LIN {X 0,Y 421.12,Z 160.701,A -85,B 0,C 180,E1 -10145.341,E2 -10145.341} C_VEL
LIN {X 0,Y 421.143,Z 165.944,A -85,B 0,C 180,E1 -10146.39,E2 -10146.39} C_VEL
LIN {X 0,Y 419.835,Z 185.67,A -85,B 0,C 180,E1 -10150.217,E2 -10150.217} C_VEL
LIN {X 0,Y 419.588,Z 189.326,A -85,B 0,C 180,E1 -10150.921,E2 -10150.921} C_VEL
LIN {X 0,Y 423.684,Z 215.471,A -85,B 0,C 180,E1 -10151.572,E2 -10151.572} C_VEL
LIN {X 0,Y 422.852,Z 297.887,A -85,B 0,C 180,E1 -10152.997,E2 -10152.997} C_VEL
LIN {X 0,Y 422.296,Z 311.131,A -85,B 0,C 180,E1 -10153.41,E2 -10153.41} C_VEL
LIN {X 0,Y 421.611,Z 324.403,A -85,B 0,C 180,E1 -10154.035,E2 -10154.035} C_VEL
LIN {X 0,Y 420.908,Z 335.549,A -85,B 0,C 180,E1 -10154.753,E2 -10154.753} C_VEL
LIN {X 0,Y 420.13,Z 347.243,A -85,B 0,C 180,E1 -10155.724,E2 -10155.724} C_VEL
LIN {X 0,Y 419.409,Z 357.602,A -85,B 0,C 180,E1 -10156.802,E2 -10156.802} C_VEL
LIN {X 0,Y 418.836,Z 366.15,A -85,B 0,C 180,E1 -10157.892,E2 -10157.892} C_VEL
LIN {X 0,Y 418.209,Z 374.037,A -85,B 0,C 180,E1 -10159.102,E2 -10159.102} C_VEL
LIN {X 0,Y 417.71,Z 381.744,A -85,B 0,C 180,E1 -10160.558,E2 -10160.558} C_VEL
LIN {X 0,Y 417.328,Z 388.855,A -85,B 0,C 180,E1 -10162.257,E2 -10162.257} C_VEL
LIN {X 0,Y 417.119,Z 393.75,A -85,B 0,C 180,E1 -10163.767,E2 -10163.767} C_VEL
LIN {X 0,Y 417.102,Z 397.206,A -85,B 0,C 180,E1 -10165.167,E2 -10165.167} C_VEL
LIN {X 0,Y 417.015,Z 399.07,A -85,B 0,C 180,E1 -10166.134,E2 -10166.134} C_VEL
LIN {X 0,Y 417.032,Z 400.471,A -85,B 0,C 180,E1 -10167.102,E2 -10167.102} C_VEL
LIN {X 0,Y 417.07,Z 401.471,A -85,B 0,C 180,E1 -10168.068,E2 -10168.068} C_VEL
LIN {X 0,Y 417.034,Z 402.08,A -85,B 0,C 180,E1 -10169.034,E2 -10169.034} C_VEL
LIN {X 0,Y 417.031,Z 402.296,A -85,B 0,C 180,E1 -10169.999,E2 -10169.999} C_VEL
LIN {X 0,Y 417.069,Z 401.469,A -85,B 0,C 180,E1 -10171.931,E2 -10171.931} C_VEL
LIN {X 0,Y 417.031,Z 400.469,A -85,B 0,C 180,E1 -10172.897,E2 -10172.897} C_VEL
LIN {X 0,Y 417.015,Z 399.066,A -85,B 0,C 180,E1 -10173.865,E2 -10173.865} C_VEL
LIN {X 0,Y 417.115,Z 396.122,A -85,B 0,C 180,E1 -10175.317,E2 -10175.317} C_VEL
LIN {X 0,Y 417.231,Z 392.136,A -85,B 0,C 180,E1 -10176.771,E2 -10176.771} C_VEL
LIN {X 0,Y 417.485,Z 386.009,A -85,B 0,C 180,E1 -10178.47,E2 -10178.47} C_VEL
LIN {X 0,Y 417.873,Z 379.318,A -85,B 0,C 180,E1 -10179.926,E2 -10179.926} C_VEL
LIN {X 0,Y 418.438,Z 371.019,A -85,B 0,C 180,E1 -10181.381,E2 -10181.381} C_VEL
LIN {X 0,Y 419.083,Z 362.518,A -85,B 0,C 180,E1 -10182.591,E2 -10182.591} C_VEL
LIN {X 0,Y 419.803,Z 352.477,A -85,B 0,C 180,E1 -10183.752,E2 -10183.752} C_VEL
LIN {X 0,Y 420.497,Z 341.624,A -85,B 0,C 180,E1 -10184.766,E2 -10184.766} C_VEL
LIN {X 0,Y 421.248,Z 330.238,A -85,B 0,C 180,E1 -10185.606,E2 -10185.606} C_VEL
LIN {X 0,Y 421.911,Z 318.552,A -85,B 0,C 180,E1 -10186.263,E2 -10186.263} C_VEL
LIN {X 0,Y 422.541,Z 306.004,A -85,B 0,C 180,E1 -10186.766,E2 -10186.766} C_VEL
LIN {X 0,Y 422.933,Z 293.279,A -85,B 0,C 180,E1 -10187.092,E2 -10187.092} C_VEL
LIN {X 0,Y 423.594,Z 214.784,A -85,B 0,C 180,E1 -10188.436,E2 -10188.436} C_VEL
LIN {X 0,Y 419.587,Z 189.324,A -85,B 0,C 180,E1 -10189.072,E2 -10189.072} C_VEL
LIN {X 0,Y 420.757,Z 171.129,A -85,B 0,C 180,E1 -10192.592,E2 -10192.592} C_VEL
LIN {X 0,Y 421.281,Z 161.977,A -85,B 0,C 180,E1 -10194.386,E2 -10194.386} C_VEL
LIN {X 0,Y 419.312,Z 151.398,A -85,B 0,C 180,E1 -10196.637,E2 -10196.637} C_VEL
LIN {X 0,Y 418.285,Z 146.379,A -85,B 0,C 180,E1 -10197.751,E2 -10197.751} C_VEL
LIN {X 0,Y 418.236,Z 146.389,A -85,B 0,C 180,E1 -10201.018,E2 -10201.018} C_VEL
LIN {X 0,Y 418.229,Z 146.39,A -85,B 0,C 180,E1 -10203.678,E2 -10203.678} C_VEL
LIN {X 0,Y 418.234,Z 146.389,A -85,B 0,C 180,E1 -10207.223,E2 -10207.223} C_VEL
LIN {X 0,Y 418.203,Z 146.39,A -85,B 0,C 180,E1 -10210.866,E2 -10210.866} C_VEL
LIN {X 0,Y 418.199,Z 146.39,A -85,B 0,C 180,E1 -10213.728,E2 -10213.728} C_VEL
LIN {X 0,Y 418.194,Z 146.389,A -85,B 0,C 180,E1 -10216.447,E2 -10216.447} C_VEL
LIN {X 0,Y 418.204,Z 146.395,A -85,B 0,C 180,E1 -10219.131,E2 -10219.131} C_VEL
LIN {X 0,Y 418.231,Z 146.389,A -85,B 0,C 180,E1 -10222.775,E2 -10222.775} C_VEL
LIN {X 0,Y 418.225,Z 146.386,A -85,B 0,C 180,E1 -10226.321,E2 -10226.321} C_VEL
LIN {X 0,Y 418.231,Z 146.384,A -85,B 0,C 180,E1 -10229.727,E2 -10229.727} C_VEL
LIN {X 0,Y 418.203,Z 146.392,A -85,B 0,C 180,E1 -10233.016,E2 -10233.016} C_VEL
LIN {X 0,Y 418.249,Z 146.385,A -85,B 0,C 180,E1 -10236.216,E2 -10236.216} C_VEL
LIN {X 0,Y 418.237,Z 146.384,A -85,B 0,C 180,E1 -10239.336,E2 -10239.336} C_VEL
LIN {X 0,Y 418.237,Z 146.39,A -85,B 0,C 180,E1 -10242.394,E2 -10242.394} C_VEL
LIN {X 0,Y 418.267,Z 146.38,A -85,B 0,C 180,E1 -10245.402,E2 -10245.402} C_VEL
LIN {X 0,Y 418.292,Z 146.383,A -85,B 0,C 180,E1 -10248.368,E2 -10248.368} C_VEL
LIN {X 0,Y 418.436,Z 146.365,A -85,B 0,C 180,E1 -10252.278,E2 -10252.278} C_VEL
LIN {X 0,Y 418.458,Z 146.362,A -85,B 0,C 180,E1 -10254.217,E2 -10254.217} C_VEL
LIN {X 0,Y 418.522,Z 146.355,A -85,B 0,C 180,E1 -10258.075,E2 -10258.075} C_VEL
LIN {X 0,Y 418.396,Z 146.364,A -85,B 0,C 180,E1 -10260.963,E2 -10260.963} C_VEL
LIN {X 0,Y 418.459,Z 146.356,A -85,B 0,C 180,E1 -10262.888,E2 -10262.888} C_VEL
LIN {X 0,Y 418.432,Z 146.36,A -85,B 0,C 180,E1 -10266.46,E2 -10266.46} C_VEL
LIN {X 0,Y 418.367,Z 146.367,A -85,B 0,C 180,E1 -10268.696,E2 -10268.696} C_VEL
LIN {X 0,Y 418.304,Z 146.383,A -85,B 0,C 180,E1 -10271.631,E2 -10271.631} C_VEL
LIN {X 0,Y 418.268,Z 146.38,A -85,B 0,C 180,E1 -10274.598,E2 -10274.598} C_VEL
LIN {X 0,Y 418.246,Z 146.388,A -85,B 0,C 180,E1 -10277.606,E2 -10277.606} C_VEL
LIN {X 0,Y 418.24,Z 146.384,A -85,B 0,C 180,E1 -10280.664,E2 -10280.664} C_VEL
LIN {X 0,Y 418.25,Z 146.384,A -85,B 0,C 180,E1 -10283.784,E2 -10283.784} C_VEL
LIN {X 0,Y 418.21,Z 146.392,A -85,B 0,C 180,E1 -10287.046,E2 -10287.046} C_VEL
LIN {X 0,Y 418.234,Z 146.384,A -85,B 0,C 180,E1 -10290.273,E2 -10290.273} C_VEL
LIN {X 0,Y 418.226,Z 146.386,A -85,B 0,C 180,E1 -10293.679,E2 -10293.679} C_VEL
LIN {X 0,Y 418.233,Z 146.388,A -85,B 0,C 180,E1 -10297.225,E2 -10297.225} C_VEL
LIN {X 0,Y 418.205,Z 146.394,A -85,B 0,C 180,E1 -10300.869,E2 -10300.869} C_VEL
LIN {X 0,Y 418.199,Z 146.388,A -85,B 0,C 180,E1 -10303.729,E2 -10303.729} C_VEL
LIN {X 0,Y 418.203,Z 146.392,A -85,B 0,C 180,E1 -10306.449,E2 -10306.449} C_VEL
LIN {X 0,Y 418.213,Z 146.388,A -85,B 0,C 180,E1 -10309.132,E2 -10309.132} C_VEL
LIN {X 0,Y 418.218,Z 146.389,A -85,B 0,C 180,E1 -10312.169,E2 -10312.169} C_VEL
LIN {X 0,Y 418.263,Z 146.38,A -85,B 0,C 180,E1 -10315.421,E2 -10315.421} C_VEL
LIN {X 0,Y 418.21,Z 146.391,A -85,B 0,C 180,E1 -10318.605,E2 -10318.605} C_VEL
LIN {X 0,Y 418.241,Z 146.387,A -85,B 0,C 180,E1 -10321.934,E2 -10321.934} C_VEL
LIN {X 0,Y 418.253,Z 146.382,A -85,B 0,C 180,E1 -10325.161,E2 -10325.161} C_VEL
LIN {X 0,Y 418.274,Z 146.556,A -85,B 0,C 180,E1 -10327.66,E2 -10327.66} C_VEL
LIN {X 0,Y 420.194,Z 156.495,A -85,B 0,C 180,E1 -10330.03,E2 -10330.03} C_VEL
LIN {X 0,Y 420.055,Z 160.959,A -85,B 0,C 180,E1 -10331.01,E2 -10331.01} C_VEL
LIN {X 0,Y 424.093,Z 181.216,A -85,B 0,C 180,E1 -10331.558,E2 -10331.558} C_VEL
LIN {X 0,Y 423.051,Z 267.557,A -85,B 0,C 180,E1 -10333.037,E2 -10333.037} C_VEL
LIN {X 0,Y 422.732,Z 281.057,A -85,B 0,C 180,E1 -10333.459,E2 -10333.459} C_VEL
LIN {X 0,Y 422.184,Z 293.856,A -85,B 0,C 180,E1 -10334.058,E2 -10334.058} C_VEL
LIN {X 0,Y 421.531,Z 305.213,A -85,B 0,C 180,E1 -10334.777,E2 -10334.777} C_VEL
LIN {X 0,Y 420.921,Z 316.902,A -85,B 0,C 180,E1 -10335.747,E2 -10335.747} C_VEL
LIN {X 0,Y 420.246,Z 327.312,A -85,B 0,C 180,E1 -10336.83,E2 -10336.83} C_VEL
LIN {X 0,Y 419.539,Z 335.854,A -85,B 0,C 180,E1 -10337.914,E2 -10337.914} C_VEL
LIN {X 0,Y 418.928,Z 343.718,A -85,B 0,C 180,E1 -10339.122,E2 -10339.122} C_VEL
LIN {X 0,Y 418.35,Z 351.403,A -85,B 0,C 180,E1 -10340.574,E2 -10340.574} C_VEL
LIN {X 0,Y 418.307,Z 351.96,A -85,B 0,C 180,E1 -10340.695,E2 -10340.695} C_VEL
LIN {X 0,Y 417.433,Z 355.07,A -85,B 0,C 180,E1 -10341.378,E2 -10341.378} C_VEL
LIN {X 0,Y 414.293,Z 359.681,A -85,B 0,C 180,E1 -10342.51,E2 -10342.51} C_VEL
LIN {X 0,Y 411.176,Z 363.603,A -85,B 0,C 180,E1 -10343.699,E2 -10343.699} C_VEL
LIN {X 0,Y 410.349,Z 365.616,A -85,B 0,C 180,E1 -10344.464,E2 -10344.464} C_VEL
LIN {X 0,Y 410.161,Z 368.857,A -85,B 0,C 180,E1 -10346.071,E2 -10346.071} C_VEL
LIN {X 0,Y 410.148,Z 370.254,A -85,B 0,C 180,E1 -10347.054,E2 -10347.054} C_VEL
LIN {X 0,Y 409.964,Z 371.864,A -85,B 0,C 180,E1 -10349.018,E2 -10349.018} C_VEL
LIN {X 0,Y 409.954,Z 372.098,A -85,B 0,C 180,E1 -10350.001,E2 -10350.001} C_VEL
LIN {X 0,Y 409.964,Z 371.91,A -85,B 0,C 180,E1 -10350.983,E2 -10350.983} C_VEL
LIN {X 0,Y 410.145,Z 370.359,A -85,B 0,C 180,E1 -10352.947,E2 -10352.947} C_VEL
LIN {X 0,Y 410.147,Z 369.009,A -85,B 0,C 180,E1 -10353.931,E2 -10353.931} C_VEL
LIN {X 0,Y 410.318,Z 366.15,A -85,B 0,C 180,E1 -10355.406,E2 -10355.406} C_VEL
LIN {X 0,Y 410.543,Z 362.273,A -85,B 0,C 180,E1 -10356.883,E2 -10356.883} C_VEL
LIN {X 0,Y 410.868,Z 357.269,A -85,B 0,C 180,E1 -10358.361,E2 -10358.361} C_VEL
LIN {X 0,Y 411.439,Z 350.965,A -85,B 0,C 180,E1 -10359.836,E2 -10359.836} C_VEL
LIN {X 0,Y 412.059,Z 343.075,A -85,B 0,C 180,E1 -10361.312,E2 -10361.312} C_VEL
LIN {X 0,Y 412.689,Z 335.03,A -85,B 0,C 180,E1 -10362.541,E2 -10362.541} C_VEL
LIN {X 0,Y 413.578,Z 325.204,A -85,B 0,C 180,E1 -10363.763,E2 -10363.763} C_VEL
LIN {X 0,Y 414.261,Z 314.161,A -85,B 0,C 180,E1 -10364.869,E2 -10364.869} C_VEL
LIN {X 0,Y 414.933,Z 303.326,A -85,B 0,C 180,E1 -10365.724,E2 -10365.724} C_VEL
LIN {X 0,Y 415.547,Z 291.357,A -85,B 0,C 180,E1 -10366.457,E2 -10366.457} C_VEL
LIN {X 0,Y 416.066,Z 278.207,A -85,B 0,C 180,E1 -10367.036,E2 -10367.036} C_VEL
LIN {X 0,Y 416.484,Z 264.956,A -85,B 0,C 180,E1 -10367.398,E2 -10367.398} C_VEL
LIN {X 0,Y 417.353,Z 181.348,A -85,B 0,C 180,E1 -10368.852,E2 -10368.852} C_VEL
LIN {X 0,Y 413.161,Z 161.121,A -85,B 0,C 180,E1 -10369.44,E2 -10369.44} C_VEL
LIN {X 0,Y 413.177,Z 157.551,A -85,B 0,C 180,E1 -10370.242,E2 -10370.242} C_VEL
LIN {X 0,Y 411.205,Z 147.261,A -85,B 0,C 180,E1 -10372.755,E2 -10372.755} C_VEL
LIN {X 0,Y 411.199,Z 147.263,A -85,B 0,C 180,E1 -10375.296,E2 -10375.296} C_VEL
LIN {X 0,Y 411.196,Z 147.261,A -85,B 0,C 180,E1 -10378.592,E2 -10378.592} C_VEL
LIN {X 0,Y 411.168,Z 147.268,A -85,B 0,C 180,E1 -10381.997,E2 -10381.997} C_VEL
LIN {X 0,Y 411.212,Z 147.259,A -85,B 0,C 180,E1 -10384.878,E2 -10384.878} C_VEL
LIN {X 0,Y 411.196,Z 147.262,A -85,B 0,C 180,E1 -10388.166,E2 -10388.166} C_VEL
LIN {X 0,Y 411.17,Z 147.267,A -85,B 0,C 180,E1 -10391.806,E2 -10391.806} C_VEL
LIN {X 0,Y 411.176,Z 147.268,A -85,B 0,C 180,E1 -10395.509,E2 -10395.509} C_VEL
LIN {X 0,Y 411.154,Z 147.268,A -85,B 0,C 180,E1 -10398.773,E2 -10398.773} C_VEL
LIN {X 0,Y 411.186,Z 147.262,A -85,B 0,C 180,E1 -10402.025,E2 -10402.025} C_VEL
LIN {X 0,Y 411.191,Z 147.262,A -85,B 0,C 180,E1 -10405.665,E2 -10405.665} C_VEL
LIN {X 0,Y 411.186,Z 147.267,A -85,B 0,C 180,E1 -10409.152,E2 -10409.152} C_VEL
LIN {X 0,Y 411.178,Z 147.265,A -85,B 0,C 180,E1 -10411.407,E2 -10411.407} C_VEL
LIN {X 0,Y 411.225,Z 147.263,A -85,B 0,C 180,E1 -10414.929,E2 -10414.929} C_VEL
LIN {X 0,Y 411.203,Z 147.26,A -85,B 0,C 180,E1 -10417.913,E2 -10417.913} C_VEL
LIN {X 0,Y 411.212,Z 147.261,A -85,B 0,C 180,E1 -10421.051,E2 -10421.051} C_VEL
LIN {X 0,Y 411.208,Z 147.262,A -85,B 0,C 180,E1 -10424.13,E2 -10424.13} C_VEL
LIN {X 0,Y 411.301,Z 147.248,A -85,B 0,C 180,E1 -10427.165,E2 -10427.165} C_VEL
LIN {X 0,Y 411.285,Z 147.254,A -85,B 0,C 180,E1 -10430.161,E2 -10430.161} C_VEL
LIN {X 0,Y 411.387,Z 147.237,A -85,B 0,C 180,E1 -10433.132,E2 -10433.132} C_VEL
LIN {X 0,Y 411.281,Z 147.25,A -85,B 0,C 180,E1 -10435.099,E2 -10435.099} C_VEL
LIN {X 0,Y 411.498,Z 147.229,A -85,B 0,C 180,E1 -10438.042,E2 -10438.042} C_VEL
LIN {X 0,Y 411.373,Z 147.239,A -85,B 0,C 180,E1 -10440.979,E2 -10440.979} C_VEL
LIN {X 0,Y 411.422,Z 147.233,A -85,B 0,C 180,E1 -10442.937,E2 -10442.937} C_VEL
LIN {X 0,Y 411.386,Z 147.237,A -85,B 0,C 180,E1 -10446.868,E2 -10446.868} C_VEL
LIN {X 0,Y 411.27,Z 147.258,A -85,B 0,C 180,E1 -10449.839,E2 -10449.839} C_VEL
LIN {X 0,Y 411.297,Z 147.249,A -85,B 0,C 180,E1 -10453.1,E2 -10453.1} C_VEL
LIN {X 0,Y 411.204,Z 147.26,A -85,B 0,C 180,E1 -10456.891,E2 -10456.891} C_VEL
LIN {X 0,Y 411.201,Z 147.262,A -85,B 0,C 180,E1 -10459.988,E2 -10459.988} C_VEL
LIN {X 0,Y 411.182,Z 147.266,A -85,B 0,C 180,E1 -10463.149,E2 -10463.149} C_VEL
LIN {X 0,Y 411.168,Z 147.264,A -85,B 0,C 180,E1 -10466.386,E2 -10466.386} C_VEL
LIN {X 0,Y 411.19,Z 147.263,A -85,B 0,C 180,E1 -10469.714,E2 -10469.714} C_VEL
LIN {X 0,Y 411.202,Z 147.267,A -85,B 0,C 180,E1 -10473.156,E2 -10473.156} C_VEL
LIN {X 0,Y 411.19,Z 147.263,A -85,B 0,C 180,E1 -10476.552,E2 -10476.552} C_VEL
LIN {X 0,Y 411.177,Z 147.263,A -85,B 0,C 180,E1 -10479.722,E2 -10479.722} C_VEL
LIN {X 0,Y 411.161,Z 147.269,A -85,B 0,C 180,E1 -10483.135,E2 -10483.135} C_VEL
LIN {X 0,Y 411.163,Z 147.265,A -85,B 0,C 180,E1 -10485.882,E2 -10485.882} C_VEL
LIN {X 0,Y 411.158,Z 147.266,A -85,B 0,C 180,E1 -10489.493,E2 -10489.493} C_VEL
LIN {X 0,Y 411.186,Z 147.263,A -85,B 0,C 180,E1 -10492.025,E2 -10492.025} C_VEL
LIN {X 0,Y 411.203,Z 147.261,A -85,B 0,C 180,E1 -10495.123,E2 -10495.123} C_VEL
LIN {X 0,Y 411.165,Z 147.267,A -85,B 0,C 180,E1 -10498.003,E2 -10498.003} C_VEL
LIN {X 0,Y 411.208,Z 147.263,A -85,B 0,C 180,E1 -10501.409,E2 -10501.409} C_VEL
LIN {X 0,Y 411.247,Z 147.354,A -85,B 0,C 180,E1 -10502.003,E2 -10502.003} C_VEL
LIN {X 0,Y 413.892,Z 160.426,A -85,B 0,C 180,E1 -10504.88,E2 -10504.88} C_VEL
LIN {X 0,Y 414.376,Z 164.377,A -85,B 0,C 180,E1 -10505.714,E2 -10505.714} C_VEL
LIN {X 0,Y 413.094,Z 182.725,A -85,B 0,C 180,E1 -10509.345,E2 -10509.345} C_VEL
LIN {X 0,Y 412.722,Z 188.983,A -85,B 0,C 180,E1 -10510.574,E2 -10510.574} C_VEL
LIN {X 0,Y 416.867,Z 215.868,A -85,B 0,C 180,E1 -10511.271,E2 -10511.271} C_VEL
LIN {X 0,Y 416.082,Z 297.641,A -85,B 0,C 180,E1 -10512.712,E2 -10512.712} C_VEL
LIN {X 0,Y 415.506,Z 310.88,A -85,B 0,C 180,E1 -10513.131,E2 -10513.131} C_VEL
LIN {X 0,Y 414.782,Z 324.149,A -85,B 0,C 180,E1 -10513.765,E2 -10513.765} C_VEL
LIN {X 0,Y 414.045,Z 335.293,A -85,B 0,C 180,E1 -10514.494,E2 -10514.494} C_VEL
LIN {X 0,Y 413.22,Z 346.897,A -85,B 0,C 180,E1 -10515.471,E2 -10515.471} C_VEL
LIN {X 0,Y 412.483,Z 357.345,A -85,B 0,C 180,E1 -10516.576,E2 -10516.576} C_VEL
LIN {X 0,Y 411.875,Z 365.893,A -85,B 0,C 180,E1 -10517.684,E2 -10517.684} C_VEL
LIN {X 0,Y 411.209,Z 373.778,A -85,B 0,C 180,E1 -10518.914,E2 -10518.914} C_VEL
LIN {X 0,Y 410.665,Z 381.485,A -85,B 0,C 180,E1 -10520.394,E2 -10520.394} C_VEL
LIN {X 0,Y 410.268,Z 388.596,A -85,B 0,C 180,E1 -10522.123,E2 -10522.123} C_VEL
LIN {X 0,Y 410.043,Z 393.819,A -85,B 0,C 180,E1 -10523.775,E2 -10523.775} C_VEL
LIN {X 0,Y 410.009,Z 396.947,A -85,B 0,C 180,E1 -10525.083,E2 -10525.083} C_VEL
LIN {X 0,Y 409.932,Z 398.812,A -85,B 0,C 180,E1 -10526.067,E2 -10526.067} C_VEL
LIN {X 0,Y 409.997,Z 401.213,A -85,B 0,C 180,E1 -10528.035,E2 -10528.035} C_VEL
LIN {X 0,Y 409.958,Z 401.821,A -85,B 0,C 180,E1 -10529.017,E2 -10529.017} C_VEL
LIN {X 0,Y 409.952,Z 402.037,A -85,B 0,C 180,E1 -10529.999,E2 -10529.999} C_VEL
LIN {X 0,Y 409.997,Z 401.211,A -85,B 0,C 180,E1 -10531.964,E2 -10531.964} C_VEL
LIN {X 0,Y 409.932,Z 398.806,A -85,B 0,C 180,E1 -10533.932,E2 -10533.932} C_VEL
LIN {X 0,Y 410.01,Z 395.861,A -85,B 0,C 180,E1 -10535.409,E2 -10535.409} C_VEL
LIN {X 0,Y 410.164,Z 391.876,A -85,B 0,C 180,E1 -10536.888,E2 -10536.888} C_VEL
LIN {X 0,Y 410.447,Z 385.748,A -85,B 0,C 180,E1 -10538.616,E2 -10538.616} C_VEL
LIN {X 0,Y 410.864,Z 379.056,A -85,B 0,C 180,E1 -10540.097,E2 -10540.097} C_VEL
LIN {X 0,Y 411.46,Z 370.757,A -85,B 0,C 180,E1 -10541.577,E2 -10541.577} C_VEL
LIN {X 0,Y 412.109,Z 362.254,A -85,B 0,C 180,E1 -10542.808,E2 -10542.808} C_VEL
LIN {X 0,Y 412.882,Z 351.988,A -85,B 0,C 180,E1 -10544.012,E2 -10544.012} C_VEL
LIN {X 0,Y 413.614,Z 341.36,A -85,B 0,C 180,E1 -10545.017,E2 -10545.017} C_VEL
LIN {X 0,Y 414.402,Z 329.974,A -85,B 0,C 180,E1 -10545.87,E2 -10545.87} C_VEL
LIN {X 0,Y 415.099,Z 318.286,A -85,B 0,C 180,E1 -10546.537,E2 -10546.537} C_VEL
LIN {X 0,Y 415.762,Z 305.736,A -85,B 0,C 180,E1 -10547.047,E2 -10547.047} C_VEL
LIN {X 0,Y 416.152,Z 293.003,A -85,B 0,C 180,E1 -10547.379,E2 -10547.379} C_VEL
LIN {X 0,Y 416.854,Z 215.725,A -85,B 0,C 180,E1 -10548.724,E2 -10548.724} C_VEL
LIN {X 0,Y 412.718,Z 189.239,A -85,B 0,C 180,E1 -10549.392,E2 -10549.392} C_VEL
LIN {X 0,Y 413.902,Z 170.865,A -85,B 0,C 180,E1 -10552.987,E2 -10552.987} C_VEL
LIN {X 0,Y 414.309,Z 163.019,A -85,B 0,C 180,E1 -10554.556,E2 -10554.556} C_VEL
LIN {X 0,Y 411.935,Z 150.593,A -85,B 0,C 180,E1 -10557.261,E2 -10557.261} C_VEL
LIN {X 0,Y 411.256,Z 147.256,A -85,B 0,C 180,E1 -10558.03,E2 -10558.03} C_VEL
LIN {X 0,Y 411.179,Z 147.269,A -85,B 0,C 180,E1 -10561.282,E2 -10561.282} C_VEL
LIN {X 0,Y 411.189,Z 147.262,A -85,B 0,C 180,E1 -10564.334,E2 -10564.334} C_VEL
LIN {X 0,Y 411.185,Z 147.263,A -85,B 0,C 180,E1 -10566.741,E2 -10566.741} C_VEL
LIN {X 0,Y 411.165,Z 147.268,A -85,B 0,C 180,E1 -10569.719,E2 -10569.719} C_VEL
LIN {X 0,Y 411.16,Z 147.271,A -85,B 0,C 180,E1 -10573.134,E2 -10573.134} C_VEL
LIN {X 0,Y 411.158,Z 147.266,A -85,B 0,C 180,E1 -10575.881,E2 -10575.881} C_VEL
LIN {X 0,Y 411.156,Z 147.268,A -85,B 0,C 180,E1 -10579.493,E2 -10579.493} C_VEL
LIN {X 0,Y 411.18,Z 147.263,A -85,B 0,C 180,E1 -10582.025,E2 -10582.025} C_VEL
LIN {X 0,Y 411.195,Z 147.266,A -85,B 0,C 180,E1 -10585.123,E2 -10585.123} C_VEL
LIN {X 0,Y 411.155,Z 147.266,A -85,B 0,C 180,E1 -10588.002,E2 -10588.002} C_VEL
LIN {X 0,Y 411.167,Z 147.265,A -85,B 0,C 180,E1 -10591.406,E2 -10591.406} C_VEL
LIN {X 0,Y 411.179,Z 147.267,A -85,B 0,C 180,E1 -10594.941,E2 -10594.941} C_VEL
LIN {X 0,Y 411.193,Z 147.262,A -85,B 0,C 180,E1 -10597.913,E2 -10597.913} C_VEL
LIN {X 0,Y 411.201,Z 147.262,A -85,B 0,C 180,E1 -10601.05,E2 -10601.05} C_VEL
LIN {X 0,Y 411.199,Z 147.264,A -85,B 0,C 180,E1 -10604.13,E2 -10604.13} C_VEL
LIN {X 0,Y 411.292,Z 147.249,A -85,B 0,C 180,E1 -10607.165,E2 -10607.165} C_VEL
LIN {X 0,Y 411.265,Z 147.258,A -85,B 0,C 180,E1 -10610.161,E2 -10610.161} C_VEL
LIN {X 0,Y 411.379,Z 147.238,A -85,B 0,C 180,E1 -10613.132,E2 -10613.132} C_VEL
LIN {X 0,Y 411.274,Z 147.251,A -85,B 0,C 180,E1 -10615.099,E2 -10615.099} C_VEL
LIN {X 0,Y 411.491,Z 147.231,A -85,B 0,C 180,E1 -10618.043,E2 -10618.043} C_VEL
LIN {X 0,Y 411.366,Z 147.24,A -85,B 0,C 180,E1 -10620.979,E2 -10620.979} C_VEL
LIN {X 0,Y 411.417,Z 147.233,A -85,B 0,C 180,E1 -10622.938,E2 -10622.938} C_VEL
LIN {X 0,Y 411.382,Z 147.238,A -85,B 0,C 180,E1 -10626.456,E2 -10626.456} C_VEL
LIN {X 0,Y 411.308,Z 147.247,A -85,B 0,C 180,E1 -10628.846,E2 -10628.846} C_VEL
LIN {X 0,Y 411.273,Z 147.256,A -85,B 0,C 180,E1 -10631.833,E2 -10631.833} C_VEL
LIN {X 0,Y 411.221,Z 147.258,A -85,B 0,C 180,E1 -10634.854,E2 -10634.854} C_VEL
LIN {X 0,Y 411.204,Z 147.262,A -85,B 0,C 180,E1 -10637.917,E2 -10637.917} C_VEL
LIN {X 0,Y 411.187,Z 147.265,A -85,B 0,C 180,E1 -10641.035,E2 -10641.035} C_VEL
LIN {X 0,Y 411.183,Z 147.262,A -85,B 0,C 180,E1 -10644.218,E2 -10644.218} C_VEL
LIN {X 0,Y 411.169,Z 147.268,A -85,B 0,C 180,E1 -10647.484,E2 -10647.484} C_VEL
LIN {X 0,Y 411.189,Z 147.263,A -85,B 0,C 180,E1 -10649.714,E2 -10649.714} C_VEL
LIN {X 0,Y 411.197,Z 147.266,A -85,B 0,C 180,E1 -10653.157,E2 -10653.157} C_VEL
LIN {X 0,Y 411.186,Z 147.265,A -85,B 0,C 180,E1 -10656.553,E2 -10656.553} C_VEL
LIN {X 0,Y 411.172,Z 147.264,A -85,B 0,C 180,E1 -10659.723,E2 -10659.723} C_VEL
LIN {X 0,Y 411.159,Z 147.268,A -85,B 0,C 180,E1 -10663.136,E2 -10663.136} C_VEL
LIN {X 0,Y 411.163,Z 147.265,A -85,B 0,C 180,E1 -10665.882,E2 -10665.882} C_VEL
LIN {X 0,Y 411.154,Z 147.271,A -85,B 0,C 180,E1 -10668.774,E2 -10668.774} C_VEL
LIN {X 0,Y 411.183,Z 147.264,A -85,B 0,C 180,E1 -10672.026,E2 -10672.026} C_VEL
LIN {X 0,Y 411.203,Z 147.26,A -85,B 0,C 180,E1 -10675.667,E2 -10675.667} C_VEL
LIN {X 0,Y 411.187,Z 147.262,A -85,B 0,C 180,E1 -10679.153,E2 -10679.153} C_VEL
LIN {X 0,Y 411.185,Z 147.266,A -85,B 0,C 180,E1 -10682.518,E2 -10682.518} C_VEL
LIN {X 0,Y 411.203,Z 147.263,A -85,B 0,C 180,E1 -10685.784,E2 -10685.784} C_VEL
LIN {X 0,Y 411.219,Z 147.419,A -85,B 0,C 180,E1 -10687.405,E2 -10687.405} C_VEL
LIN {X 0,Y 413.177,Z 157.134,A -85,B 0,C 180,E1 -10689.764,E2 -10689.764} C_VEL
LIN {X 0,Y 413.163,Z 161.186,A -85,B 0,C 180,E1 -10690.675,E2 -10690.675} C_VEL
LIN {X 0,Y 417.367,Z 181.958,A -85,B 0,C 180,E1 -10691.258,E2 -10691.258} C_VEL
LIN {X 0,Y 416.27,Z 267.835,A -85,B 0,C 180,E1 -10692.753,E2 -10692.753} C_VEL
LIN {X 0,Y 415.954,Z 281.326,A -85,B 0,C 180,E1 -10693.182,E2 -10693.182} C_VEL
LIN {X 0,Y 415.365,Z 294.123,A -85,B 0,C 180,E1 -10693.789,E2 -10693.789} C_VEL
LIN {X 0,Y 414.702,Z 305.478,A -85,B 0,C 180,E1 -10694.52,E2 -10694.52} C_VEL
LIN {X 0,Y 414.102,Z 316.122,A -85,B 0,C 180,E1 -10695.406,E2 -10695.406} C_VEL
LIN {X 0,Y 413.426,Z 326.511,A -85,B 0,C 180,E1 -10696.483,E2 -10696.483} C_VEL
LIN {X 0,Y 412.604,Z 336.116,A -85,B 0,C 180,E1 -10697.707,E2 -10697.707} C_VEL
LIN {X 0,Y 411.963,Z 343.98,A -85,B 0,C 180,E1 -10698.936,E2 -10698.936} C_VEL
LIN {X 0,Y 411.36,Z 351.664,A -85,B 0,C 180,E1 -10700.412,E2 -10700.412} C_VEL
LIN {X 0,Y 410.778,Z 358.714,A -85,B 0,C 180,E1 -10702.134,E2 -10702.134} C_VEL
LIN {X 0,Y 410.551,Z 363.004,A -85,B 0,C 180,E1 -10703.472,E2 -10703.472} C_VEL
LIN {X 0,Y 410.349,Z 365.616,A -85,B 0,C 180,E1 -10704.464,E2 -10704.464} C_VEL
LIN {X 0,Y 409.542,Z 367.409,A -85,B 0,C 180,E1 -10705.243,E2 -10705.243} C_VEL
LIN {X 0,Y 406.546,Z 369.725,A -85,B 0,C 180,E1 -10706.531,E2 -10706.531} C_VEL
LIN {X 0,Y 404.071,Z 371.118,A -85,B 0,C 180,E1 -10707.587,E2 -10707.587} C_VEL
LIN {X 0,Y 402.93,Z 371.908,A -85,B 0,C 180,E1 -10708.552,E2 -10708.552} C_VEL
LIN {X 0,Y 402.902,Z 371.933,A -85,B 0,C 180,E1 -10708.692,E2 -10708.692} C_VEL
LIN {X 0,Y 402.877,Z 372.356,A -85,B 0,C 180,E1 -10710.001,E2 -10710.001} C_VEL
LIN {X 0,Y 402.89,Z 372.168,A -85,B 0,C 180,E1 -10711,E2 -10711} C_VEL
LIN {X 0,Y 403.065,Z 370.618,A -85,B 0,C 180,E1 -10712.999,E2 -10712.999} C_VEL
LIN {X 0,Y 403.059,Z 369.268,A -85,B 0,C 180,E1 -10714,E2 -10714} C_VEL
LIN {X 0,Y 403.269,Z 366.407,A -85,B 0,C 180,E1 -10715.501,E2 -10715.501} C_VEL
LIN {X 0,Y 403.486,Z 362.531,A -85,B 0,C 180,E1 -10717.004,E2 -10717.004} C_VEL
LIN {X 0,Y 403.854,Z 357.527,A -85,B 0,C 180,E1 -10718.507,E2 -10718.507} C_VEL
LIN {X 0,Y 404.455,Z 351.222,A -85,B 0,C 180,E1 -10720.007,E2 -10720.007} C_VEL
LIN {X 0,Y 405.097,Z 343.332,A -85,B 0,C 180,E1 -10721.509,E2 -10721.509} C_VEL
LIN {X 0,Y 405.768,Z 335.286,A -85,B 0,C 180,E1 -10722.758,E2 -10722.758} C_VEL
LIN {X 0,Y 406.704,Z 325.459,A -85,B 0,C 180,E1 -10724.001,E2 -10724.001} C_VEL
LIN {X 0,Y 407.3,Z 315.798,A -85,B 0,C 180,E1 -10725.001,E2 -10725.001} C_VEL
LIN {X 0,Y 408.028,Z 305.336,A -85,B 0,C 180,E1 -10725.869,E2 -10725.869} C_VEL
LIN {X 0,Y 408.67,Z 293.859,A -85,B 0,C 180,E1 -10726.613,E2 -10726.613} C_VEL
LIN {X 0,Y 409.225,Z 280.878,A -85,B 0,C 180,E1 -10727.233,E2 -10727.233} C_VEL
LIN {X 0,Y 409.642,Z 268.165,A -85,B 0,C 180,E1 -10727.633,E2 -10727.633} C_VEL
LIN {X 0,Y 410.612,Z 182.102,A -85,B 0,C 180,E1 -10729.164,E2 -10729.164} C_VEL
LIN {X 0,Y 406.301,Z 161.329,A -85,B 0,C 180,E1 -10729.791,E2 -10729.791} C_VEL
LIN {X 0,Y 405.821,Z 156.281,A -85,B 0,C 180,E1 -10730.979,E2 -10730.979} C_VEL
LIN {X 0,Y 404.18,Z 148.135,A -85,B 0,C 180,E1 -10733.041,E2 -10733.041} C_VEL
LIN {X 0,Y 404.152,Z 148.144,A -85,B 0,C 180,E1 -10735.769,E2 -10735.769} C_VEL
LIN {X 0,Y 404.159,Z 148.138,A -85,B 0,C 180,E1 -10739.137,E2 -10739.137} C_VEL
LIN {X 0,Y 404.143,Z 148.139,A -85,B 0,C 180,E1 -10742.622,E2 -10742.622} C_VEL
LIN {X 0,Y 404.182,Z 148.137,A -85,B 0,C 180,E1 -10745.19,E2 -10745.19} C_VEL
LIN {X 0,Y 404.135,Z 148.141,A -85,B 0,C 180,E1 -10748.759,E2 -10748.759} C_VEL
LIN {X 0,Y 404.114,Z 148.148,A -85,B 0,C 180,E1 -10751.598,E2 -10751.598} C_VEL
LIN {X 0,Y 404.145,Z 148.139,A -85,B 0,C 180,E1 -10754.522,E2 -10754.522} C_VEL
LIN {X 0,Y 404.131,Z 148.148,A -85,B 0,C 180,E1 -10757.295,E2 -10757.295} C_VEL
LIN {X 0,Y 404.132,Z 148.141,A -85,B 0,C 180,E1 -10759.951,E2 -10759.951} C_VEL
LIN {X 0,Y 404.134,Z 148.148,A -85,B 0,C 180,E1 -10763.125,E2 -10763.125} C_VEL
LIN {X 0,Y 404.137,Z 148.14,A -85,B 0,C 180,E1 -10766.187,E2 -10766.187} C_VEL
LIN {X 0,Y 404.142,Z 148.14,A -85,B 0,C 180,E1 -10769.714,E2 -10769.714} C_VEL
LIN {X 0,Y 404.126,Z 148.145,A -85,B 0,C 180,E1 -10773.118,E2 -10773.118} C_VEL
LIN {X 0,Y 404.161,Z 148.14,A -85,B 0,C 180,E1 -10776.425,E2 -10776.425} C_VEL
LIN {X 0,Y 404.19,Z 148.134,A -85,B 0,C 180,E1 -10779.874,E2 -10779.874} C_VEL
LIN {X 0,Y 404.172,Z 148.138,A -85,B 0,C 180,E1 -10783.013,E2 -10783.013} C_VEL
LIN {X 0,Y 404.281,Z 148.124,A -85,B 0,C 180,E1 -10786.939,E2 -10786.939} C_VEL
LIN {X 0,Y 404.251,Z 148.129,A -85,B 0,C 180,E1 -10789.988,E2 -10789.988} C_VEL
LIN {X 0,Y 404.337,Z 148.116,A -85,B 0,C 180,E1 -10793.011,E2 -10793.011} C_VEL
LIN {X 0,Y 404.253,Z 148.126,A -85,B 0,C 180,E1 -10795.013,E2 -10795.013} C_VEL
LIN {X 0,Y 404.467,Z 148.104,A -85,B 0,C 180,E1 -10798.008,E2 -10798.008} C_VEL
LIN {X 0,Y 404.343,Z 148.114,A -85,B 0,C 180,E1 -10800.996,E2 -10800.996} C_VEL
LIN {X 0,Y 404.355,Z 148.113,A -85,B 0,C 180,E1 -10802.989,E2 -10802.989} C_VEL
LIN {X 0,Y 404.362,Z 148.118,A -85,B 0,C 180,E1 -10805.986,E2 -10805.986} C_VEL
LIN {X 0,Y 404.251,Z 148.126,A -85,B 0,C 180,E1 -10809.002,E2 -10809.002} C_VEL
LIN {X 0,Y 404.24,Z 148.131,A -85,B 0,C 180,E1 -10812.042,E2 -10812.042} C_VEL
LIN {X 0,Y 404.153,Z 148.14,A -85,B 0,C 180,E1 -10815.12,E2 -10815.12} C_VEL
LIN {X 0,Y 404.132,Z 148.141,A -85,B 0,C 180,E1 -10818.242,E2 -10818.242} C_VEL
LIN {X 0,Y 404.127,Z 148.148,A -85,B 0,C 180,E1 -10821.42,E2 -10821.42} C_VEL
LIN {X 0,Y 404.132,Z 148.141,A -85,B 0,C 180,E1 -10824.669,E2 -10824.669} C_VEL
LIN {X 0,Y 404.098,Z 148.145,A -85,B 0,C 180,E1 -10828.007,E2 -10828.007} C_VEL
LIN {X 0,Y 404.137,Z 148.14,A -85,B 0,C 180,E1 -10830.286,E2 -10830.286} C_VEL
LIN {X 0,Y 404.136,Z 148.141,A -85,B 0,C 180,E1 -10833.813,E2 -10833.813} C_VEL
LIN {X 0,Y 404.133,Z 148.146,A -85,B 0,C 180,E1 -10836.875,E2 -10836.875} C_VEL
LIN {X 0,Y 404.116,Z 148.143,A -85,B 0,C 180,E1 -10840.075,E2 -10840.075} C_VEL
LIN {X 0,Y 404.141,Z 148.144,A -85,B 0,C 180,E1 -10843.082,E2 -10843.082} C_VEL
LIN {X 0,Y 404.12,Z 148.142,A -85,B 0,C 180,E1 -10845.922,E2 -10845.922} C_VEL
LIN {X 0,Y 404.102,Z 148.151,A -85,B 0,C 180,E1 -10848.633,E2 -10848.633} C_VEL
LIN {X 0,Y 404.14,Z 148.14,A -85,B 0,C 180,E1 -10851.495,E2 -10851.495} C_VEL
LIN {X 0,Y 404.178,Z 148.137,A -85,B 0,C 180,E1 -10854.983,E2 -10854.983} C_VEL
LIN {X 0,Y 404.14,Z 148.147,A -85,B 0,C 180,E1 -10858.442,E2 -10858.442} C_VEL
LIN {X 0,Y 404.212,Z 148.234,A -85,B 0,C 180,E1 -10861.719,E2 -10861.719} C_VEL
LIN {X 0,Y 406.912,Z 161.47,A -85,B 0,C 180,E1 -10864.693,E2 -10864.693} C_VEL
LIN {X 0,Y 407.443,Z 165.423,A -85,B 0,C 180,E1 -10865.545,E2 -10865.545} C_VEL
LIN {X 0,Y 406.227,Z 182.538,A -85,B 0,C 180,E1 -10868.995,E2 -10868.995} C_VEL
LIN {X 0,Y 405.787,Z 188.8,A -85,B 0,C 180,E1 -10870.245,E2 -10870.245} C_VEL
LIN {X 0,Y 410.171,Z 216.788,A -85,B 0,C 180,E1 -10870.975,E2 -10870.975} C_VEL
LIN {X 0,Y 409.312,Z 297.394,A -85,B 0,C 180,E1 -10872.417,E2 -10872.417} C_VEL
LIN {X 0,Y 408.722,Z 310.629,A -85,B 0,C 180,E1 -10872.842,E2 -10872.842} C_VEL
LIN {X 0,Y 407.965,Z 323.896,A -85,B 0,C 180,E1 -10873.486,E2 -10873.486} C_VEL
LIN {X 0,Y 407.205,Z 335.038,A -85,B 0,C 180,E1 -10874.226,E2 -10874.226} C_VEL
LIN {X 0,Y 406.319,Z 346.64,A -85,B 0,C 180,E1 -10875.219,E2 -10875.219} C_VEL
LIN {X 0,Y 405.606,Z 356.667,A -85,B 0,C 180,E1 -10876.294,E2 -10876.294} C_VEL
LIN {X 0,Y 404.916,Z 365.635,A -85,B 0,C 180,E1 -10877.469,E2 -10877.469} C_VEL
LIN {X 0,Y 404.19,Z 373.519,A -85,B 0,C 180,E1 -10878.719,E2 -10878.719} C_VEL
LIN {X 0,Y 403.627,Z 381.226,A -85,B 0,C 180,E1 -10880.225,E2 -10880.225} C_VEL
LIN {X 0,Y 403.203,Z 388.336,A -85,B 0,C 180,E1 -10881.984,E2 -10881.984} C_VEL
LIN {X 0,Y 402.963,Z 393.069,A -85,B 0,C 180,E1 -10883.491,E2 -10883.491} C_VEL
LIN {X 0,Y 402.918,Z 396.688,A -85,B 0,C 180,E1 -10884.996,E2 -10884.996} C_VEL
LIN {X 0,Y 402.852,Z 398.553,A -85,B 0,C 180,E1 -10885.998,E2 -10885.998} C_VEL
LIN {X 0,Y 402.907,Z 400.954,A -85,B 0,C 180,E1 -10888,E2 -10888} C_VEL
LIN {X 0,Y 402.884,Z 401.563,A -85,B 0,C 180,E1 -10889,E2 -10889} C_VEL
LIN {X 0,Y 402.875,Z 401.779,A -85,B 0,C 180,E1 -10889.999,E2 -10889.999} C_VEL
LIN {X 0,Y 402.883,Z 401.561,A -85,B 0,C 180,E1 -10890.999,E2 -10890.999} C_VEL
LIN {X 0,Y 402.907,Z 400.951,A -85,B 0,C 180,E1 -10891.999,E2 -10891.999} C_VEL
LIN {X 0,Y 402.852,Z 398.547,A -85,B 0,C 180,E1 -10894.001,E2 -10894.001} C_VEL
LIN {X 0,Y 402.906,Z 395.6,A -85,B 0,C 180,E1 -10895.505,E2 -10895.505} C_VEL
LIN {X 0,Y 403.076,Z 391.614,A -85,B 0,C 180,E1 -10897.01,E2 -10897.01} C_VEL
LIN {X 0,Y 403.384,Z 385.486,A -85,B 0,C 180,E1 -10898.768,E2 -10898.768} C_VEL
LIN {X 0,Y 403.817,Z 378.793,A -85,B 0,C 180,E1 -10900.275,E2 -10900.275} C_VEL
LIN {X 0,Y 404.486,Z 370.495,A -85,B 0,C 180,E1 -10901.779,E2 -10901.779} C_VEL
LIN {X 0,Y 405.137,Z 361.99,A -85,B 0,C 180,E1 -10903.032,E2 -10903.032} C_VEL
LIN {X 0,Y 405.969,Z 351.724,A -85,B 0,C 180,E1 -10904.255,E2 -10904.255} C_VEL
LIN {X 0,Y 406.742,Z 341.096,A -85,B 0,C 180,E1 -10905.277,E2 -10905.277} C_VEL
LIN {X 0,Y 407.583,Z 329.71,A -85,B 0,C 180,E1 -10906.143,E2 -10906.143} C_VEL
LIN {X 0,Y 408.3,Z 318.02,A -85,B 0,C 180,E1 -10906.821,E2 -10906.821} C_VEL
LIN {X 0,Y 408.991,Z 305.467,A -85,B 0,C 180,E1 -10907.339,E2 -10907.339} C_VEL
LIN {X 0,Y 409.387,Z 292.728,A -85,B 0,C 180,E1 -10907.676,E2 -10907.676} C_VEL
LIN {X 0,Y 410.158,Z 216.606,A -85,B 0,C 180,E1 -10909.02,E2 -10909.02} C_VEL
LIN {X 0,Y 405.78,Z 188.95,A -85,B 0,C 180,E1 -10909.738,E2 -10909.738} C_VEL
LIN {X 0,Y 406.983,Z 171.907,A -85,B 0,C 180,E1 -10913.132,E2 -10913.132} C_VEL
LIN {X 0,Y 407.336,Z 164.059,A -85,B 0,C 180,E1 -10914.733,E2 -10914.733} C_VEL
LIN {X 0,Y 404.766,Z 150.786,A -85,B 0,C 180,E1 -10917.684,E2 -10917.684} C_VEL
LIN {X 0,Y 404.183,Z 148.139,A -85,B 0,C 180,E1 -10918.317,E2 -10918.317} C_VEL
LIN {X 0,Y 404.136,Z 148.147,A -85,B 0,C 180,E1 -10921.557,E2 -10921.557} C_VEL
LIN {X 0,Y 404.174,Z 148.137,A -85,B 0,C 180,E1 -10925.016,E2 -10925.016} C_VEL
LIN {X 0,Y 404.13,Z 148.142,A -85,B 0,C 180,E1 -10928.758,E2 -10928.758} C_VEL
LIN {X 0,Y 404.104,Z 148.148,A -85,B 0,C 180,E1 -10931.596,E2 -10931.596} C_VEL
LIN {X 0,Y 404.139,Z 148.14,A -85,B 0,C 180,E1 -10934.521,E2 -10934.521} C_VEL
LIN {X 0,Y 404.115,Z 148.148,A -85,B 0,C 180,E1 -10937.293,E2 -10937.293} C_VEL
LIN {X 0,Y 404.126,Z 148.142,A -85,B 0,C 180,E1 -10939.95,E2 -10939.95} C_VEL
LIN {X 0,Y 404.128,Z 148.147,A -85,B 0,C 180,E1 -10943.125,E2 -10943.125} C_VEL
LIN {X 0,Y 404.13,Z 148.141,A -85,B 0,C 180,E1 -10946.186,E2 -10946.186} C_VEL
LIN {X 0,Y 404.134,Z 148.14,A -85,B 0,C 180,E1 -10949.714,E2 -10949.714} C_VEL
LIN {X 0,Y 404.109,Z 148.146,A -85,B 0,C 180,E1 -10953.117,E2 -10953.117} C_VEL
LIN {X 0,Y 404.14,Z 148.144,A -85,B 0,C 180,E1 -10956.424,E2 -10956.424} C_VEL
LIN {X 0,Y 404.147,Z 148.14,A -85,B 0,C 180,E1 -10959.888,E2 -10959.888} C_VEL
LIN {X 0,Y 404.164,Z 148.138,A -85,B 0,C 180,E1 -10963.013,E2 -10963.013} C_VEL
LIN {X 0,Y 404.274,Z 148.124,A -85,B 0,C 180,E1 -10966.939,E2 -10966.939} C_VEL
LIN {X 0,Y 404.233,Z 148.132,A -85,B 0,C 180,E1 -10969.988,E2 -10969.988} C_VEL
LIN {X 0,Y 404.33,Z 148.116,A -85,B 0,C 180,E1 -10973.011,E2 -10973.011} C_VEL
LIN {X 0,Y 404.245,Z 148.127,A -85,B 0,C 180,E1 -10975.013,E2 -10975.013} C_VEL
LIN {X 0,Y 404.46,Z 148.107,A -85,B 0,C 180,E1 -10978.008,E2 -10978.008} C_VEL
LIN {X 0,Y 404.336,Z 148.115,A -85,B 0,C 180,E1 -10980.996,E2 -10980.996} C_VEL
LIN {X 0,Y 404.377,Z 148.11,A -85,B 0,C 180,E1 -10982.989,E2 -10982.989} C_VEL
LIN {X 0,Y 404.335,Z 148.116,A -85,B 0,C 180,E1 -10986.45,E2 -10986.45} C_VEL
LIN {X 0,Y 404.255,Z 148.126,A -85,B 0,C 180,E1 -10989.002,E2 -10989.002} C_VEL
LIN {X 0,Y 404.246,Z 148.129,A -85,B 0,C 180,E1 -10992.042,E2 -10992.042} C_VEL
LIN {X 0,Y 404.166,Z 148.139,A -85,B 0,C 180,E1 -10995.12,E2 -10995.12} C_VEL
LIN {X 0,Y 404.157,Z 148.138,A -85,B 0,C 180,E1 -10998.241,E2 -10998.241} C_VEL
LIN {X 0,Y 404.15,Z 148.145,A -85,B 0,C 180,E1 -11001.419,E2 -11001.419} C_VEL
LIN {X 0,Y 404.14,Z 148.141,A -85,B 0,C 180,E1 -11004.668,E2 -11004.668} C_VEL
LIN {X 0,Y 404.111,Z 148.144,A -85,B 0,C 180,E1 -11008.006,E2 -11008.006} C_VEL
LIN {X 0,Y 404.136,Z 148.14,A -85,B 0,C 180,E1 -11010.286,E2 -11010.286} C_VEL
LIN {X 0,Y 404.131,Z 148.141,A -85,B 0,C 180,E1 -11013.814,E2 -11013.814} C_VEL
LIN {X 0,Y 404.129,Z 148.147,A -85,B 0,C 180,E1 -11016.876,E2 -11016.876} C_VEL
LIN {X 0,Y 404.111,Z 148.144,A -85,B 0,C 180,E1 -11020.076,E2 -11020.076} C_VEL
LIN {X 0,Y 404.139,Z 148.143,A -85,B 0,C 180,E1 -11023.083,E2 -11023.083} C_VEL
LIN {X 0,Y 404.143,Z 148.14,A -85,B 0,C 180,E1 -11025.927,E2 -11025.927} C_VEL
LIN {X 0,Y 404.109,Z 148.15,A -85,B 0,C 180,E1 -11028.635,E2 -11028.635} C_VEL
LIN {X 0,Y 404.14,Z 148.14,A -85,B 0,C 180,E1 -11031.495,E2 -11031.495} C_VEL
LIN {X 0,Y 404.182,Z 148.136,A -85,B 0,C 180,E1 -11034.985,E2 -11034.985} C_VEL
LIN {X 0,Y 404.14,Z 148.144,A -85,B 0,C 180,E1 -11038.555,E2 -11038.555} C_VEL
LIN {X 0,Y 404.153,Z 148.139,A -85,B 0,C 180,E1 -11040.864,E2 -11040.864} C_VEL
LIN {X 0,Y 404.145,Z 148.146,A -85,B 0,C 180,E1 -11044.232,E2 -11044.232} C_VEL
LIN {X 0,Y 404.195,Z 148.33,A -85,B 0,C 180,E1 -11047.154,E2 -11047.154} C_VEL
LIN {X 0,Y 406.296,Z 158.925,A -85,B 0,C 180,E1 -11049.761,E2 -11049.761} C_VEL
LIN {X 0,Y 406.298,Z 161.441,A -85,B 0,C 180,E1 -11050.336,E2 -11050.336} C_VEL
LIN {X 0,Y 410.607,Z 182.291,A -85,B 0,C 180,E1 -11050.938,E2 -11050.938} C_VEL
LIN {X 0,Y 409.581,Z 266.638,A -85,B 0,C 180,E1 -11052.43,E2 -11052.43} C_VEL
LIN {X 0,Y 409.264,Z 279.291,A -85,B 0,C 180,E1 -11052.802,E2 -11052.802} C_VEL
LIN {X 0,Y 408.69,Z 292.136,A -85,B 0,C 180,E1 -11053.389,E2 -11053.389} C_VEL
LIN {X 0,Y 408.01,Z 303.999,A -85,B 0,C 180,E1 -11054.131,E2 -11054.131} C_VEL
LIN {X 0,Y 407.336,Z 314.753,A -85,B 0,C 180,E1 -11055.002,E2 -11055.002} C_VEL
LIN {X 0,Y 406.645,Z 325.709,A -85,B 0,C 180,E1 -11056.126,E2 -11056.126} C_VEL
LIN {X 0,Y 405.828,Z 334.606,A -85,B 0,C 180,E1 -11057.245,E2 -11057.245} C_VEL
LIN {X 0,Y 405.01,Z 344.241,A -85,B 0,C 180,E1 -11058.743,E2 -11058.743} C_VEL
LIN {X 0,Y 404.347,Z 351.925,A -85,B 0,C 180,E1 -11060.244,E2 -11060.244} C_VEL
LIN {X 0,Y 403.744,Z 358.975,A -85,B 0,C 180,E1 -11061.996,E2 -11061.996} C_VEL
LIN {X 0,Y 403.487,Z 363.552,A -85,B 0,C 180,E1 -11063.459,E2 -11063.459} C_VEL
LIN {X 0,Y 403.155,Z 367.262,A -85,B 0,C 180,E1 -11065,E2 -11065} C_VEL
LIN {X 0,Y 403.071,Z 369.118,A -85,B 0,C 180,E1 -11066.001,E2 -11066.001} C_VEL
LIN {X 0,Y 403.068,Z 370.513,A -85,B 0,C 180,E1 -11067.002,E2 -11067.002} C_VEL
LIN {X 0,Y 402.902,Z 371.933,A -85,B 0,C 180,E1 -11068.692,E2 -11068.692} C_VEL
LIN {X 0,Y 402.226,Z 372.346,A -85,B 0,C 180,E1 -11069.525,E2 -11069.525} C_VEL
LIN {X 0,Y 399.437,Z 372.458,A -85,B 0,C 180,E1 -11070.885,E2 -11070.885} C_VEL
LIN {X 0,Y 397.084,Z 371.955,A -85,B 0,C 180,E1 -11071.979,E2 -11071.979} C_VEL
LIN {X 0,Y 396.059,Z 371.165,A -85,B 0,C 180,E1 -11072.818,E2 -11072.818} C_VEL
LIN {X 0,Y 395.968,Z 370.815,A -85,B 0,C 180,E1 -11073.1,E2 -11073.1} C_VEL
LIN {X 0,Y 395.974,Z 369.527,A -85,B 0,C 180,E1 -11074.072,E2 -11074.072} C_VEL
LIN {X 0,Y 396.221,Z 366.665,A -85,B 0,C 180,E1 -11075.599,E2 -11075.599} C_VEL
LIN {X 0,Y 396.43,Z 362.789,A -85,B 0,C 180,E1 -11077.129,E2 -11077.129} C_VEL
LIN {X 0,Y 396.834,Z 357.784,A -85,B 0,C 180,E1 -11078.658,E2 -11078.658} C_VEL
LIN {X 0,Y 397.465,Z 351.479,A -85,B 0,C 180,E1 -11080.185,E2 -11080.185} C_VEL
LIN {X 0,Y 398.144,Z 343.588,A -85,B 0,C 180,E1 -11081.713,E2 -11081.713} C_VEL
LIN {X 0,Y 398.858,Z 335.542,A -85,B 0,C 180,E1 -11082.983,E2 -11082.983} C_VEL
LIN {X 0,Y 399.827,Z 325.714,A -85,B 0,C 180,E1 -11084.246,E2 -11084.246} C_VEL
LIN {X 0,Y 400.561,Z 314.669,A -85,B 0,C 180,E1 -11085.389,E2 -11085.389} C_VEL
LIN {X 0,Y 401.289,Z 303.831,A -85,B 0,C 180,E1 -11086.273,E2 -11086.273} C_VEL
LIN {X 0,Y 401.959,Z 291.858,A -85,B 0,C 180,E1 -11087.03,E2 -11087.03} C_VEL
LIN {X 0,Y 402.556,Z 278.697,A -85,B 0,C 180,E1 -11087.626,E2 -11087.626} C_VEL
LIN {X 0,Y 402.995,Z 265.43,A -85,B 0,C 180,E1 -11088,E2 -11088} C_VEL
LIN {X 0,Y 403.905,Z 183.19,A -85,B 0,C 180,E1 -11089.479,E2 -11089.479} C_VEL
LIN {X 0,Y 399.422,Z 161.663,A -85,B 0,C 180,E1 -11090.128,E2 -11090.128} C_VEL
LIN {X 0,Y 398.358,Z 155.038,A -85,B 0,C 180,E1 -11091.746,E2 -11091.746} C_VEL
LIN {X 0,Y 397.138,Z 149.013,A -85,B 0,C 180,E1 -11093.3,E2 -11093.3} C_VEL
LIN {X 0,Y 397.097,Z 149.022,A -85,B 0,C 180,E1 -11096.261,E2 -11096.261} C_VEL
LIN {X 0,Y 397.103,Z 149.023,A -85,B 0,C 180,E1 -11099.863,E2 -11099.863} C_VEL
LIN {X 0,Y 397.12,Z 149.021,A -85,B 0,C 180,E1 -11103.718,E2 -11103.718} C_VEL
LIN {X 0,Y 397.092,Z 149.02,A -85,B 0,C 180,E1 -11107.208,E2 -11107.208} C_VEL
LIN {X 0,Y 397.057,Z 149.022,A -85,B 0,C 180,E1 -11110.437,E2 -11110.437} C_VEL
LIN {X 0,Y 397.101,Z 149.021,A -85,B 0,C 180,E1 -11113.648,E2 -11113.648} C_VEL
LIN {X 0,Y 397.101,Z 149.017,A -85,B 0,C 180,E1 -11116.521,E2 -11116.521} C_VEL
LIN {X 0,Y 397.086,Z 149.019,A -85,B 0,C 180,E1 -11120.419,E2 -11120.419} C_VEL
LIN {X 0,Y 397.096,Z 149.023,A -85,B 0,C 180,E1 -11123.005,E2 -11123.005} C_VEL
LIN {X 0,Y 397.111,Z 149.019,A -85,B 0,C 180,E1 -11126.727,E2 -11126.727} C_VEL
LIN {X 0,Y 397.116,Z 149.016,A -85,B 0,C 180,E1 -11130.295,E2 -11130.295} C_VEL
LIN {X 0,Y 397.089,Z 149.018,A -85,B 0,C 180,E1 -11133.738,E2 -11133.738} C_VEL
LIN {X 0,Y 397.106,Z 149.019,A -85,B 0,C 180,E1 -11137.085,E2 -11137.085} C_VEL
LIN {X 0,Y 397.143,Z 149.015,A -85,B 0,C 180,E1 -11140.352,E2 -11140.352} C_VEL
LIN {X 0,Y 397.125,Z 149.014,A -85,B 0,C 180,E1 -11143.551,E2 -11143.551} C_VEL
LIN {X 0,Y 397.227,Z 149.005,A -85,B 0,C 180,E1 -11146.703,E2 -11146.703} C_VEL
LIN {X 0,Y 397.212,Z 149.004,A -85,B 0,C 180,E1 -11149.809,E2 -11149.809} C_VEL
LIN {X 0,Y 397.29,Z 148.994,A -85,B 0,C 180,E1 -11152.887,E2 -11152.887} C_VEL
LIN {X 0,Y 397.224,Z 149.002,A -85,B 0,C 180,E1 -11154.925,E2 -11154.925} C_VEL
LIN {X 0,Y 397.436,Z 148.98,A -85,B 0,C 180,E1 -11157.973,E2 -11157.973} C_VEL
LIN {X 0,Y 397.434,Z 148.982,A -85,B 0,C 180,E1 -11162.027,E2 -11162.027} C_VEL
LIN {X 0,Y 397.315,Z 148.995,A -85,B 0,C 180,E1 -11166.092,E2 -11166.092} C_VEL
LIN {X 0,Y 397.223,Z 149.002,A -85,B 0,C 180,E1 -11169.163,E2 -11169.163} C_VEL
LIN {X 0,Y 397.203,Z 149.005,A -85,B 0,C 180,E1 -11172.259,E2 -11172.259} C_VEL
LIN {X 0,Y 397.106,Z 149.02,A -85,B 0,C 180,E1 -11175.395,E2 -11175.395} C_VEL
LIN {X 0,Y 397.084,Z 149.019,A -85,B 0,C 180,E1 -11178.577,E2 -11178.577} C_VEL
LIN {X 0,Y 397.087,Z 149.021,A -85,B 0,C 180,E1 -11181.819,E2 -11181.819} C_VEL
LIN {X 0,Y 397.1,Z 149.021,A -85,B 0,C 180,E1 -11185.135,E2 -11185.135} C_VEL
LIN {X 0,Y 397.058,Z 149.022,A -85,B 0,C 180,E1 -11188.549,E2 -11188.549} C_VEL
LIN {X 0,Y 397.075,Z 149.021,A -85,B 0,C 180,E1 -11191.835,E2 -11191.835} C_VEL
LIN {X 0,Y 397.116,Z 149.016,A -85,B 0,C 180,E1 -11194.494,E2 -11194.494} C_VEL
LIN {X 0,Y 397.092,Z 149.018,A -85,B 0,C 180,E1 -11198.276,E2 -11198.276} C_VEL
LIN {X 0,Y 397.051,Z 149.023,A -85,B 0,C 180,E1 -11201.977,E2 -11201.977} C_VEL
LIN {X 0,Y 397.085,Z 149.022,A -85,B 0,C 180,E1 -11205.069,E2 -11205.069} C_VEL
LIN {X 0,Y 397.051,Z 149.023,A -85,B 0,C 180,E1 -11208.024,E2 -11208.024} C_VEL
LIN {X 0,Y 397.092,Z 149.018,A -85,B 0,C 180,E1 -11211.724,E2 -11211.724} C_VEL
LIN {X 0,Y 397.12,Z 149.014,A -85,B 0,C 180,E1 -11215.506,E2 -11215.506} C_VEL
LIN {X 0,Y 397.078,Z 149.023,A -85,B 0,C 180,E1 -11219.117,E2 -11219.117} C_VEL
LIN {X 0,Y 397.161,Z 149.112,A -85,B 0,C 180,E1 -11221.423,E2 -11221.423} C_VEL
LIN {X 0,Y 399.918,Z 162.513,A -85,B 0,C 180,E1 -11224.497,E2 -11224.497} C_VEL
LIN {X 0,Y 400.489,Z 167.444,A -85,B 0,C 180,E1 -11225.575,E2 -11225.575} C_VEL
LIN {X 0,Y 399.065,Z 186.014,A -85,B 0,C 180,E1 -11229.376,E2 -11229.376} C_VEL
LIN {X 0,Y 398.897,Z 188.536,A -85,B 0,C 180,E1 -11229.889,E2 -11229.889} C_VEL
LIN {X 0,Y 403.427,Z 217.351,A -85,B 0,C 180,E1 -11230.659,E2 -11230.659} C_VEL
LIN {X 0,Y 402.556,Z 297.148,A -85,B 0,C 180,E1 -11232.112,E2 -11232.112} C_VEL
LIN {X 0,Y 401.953,Z 310.379,A -85,B 0,C 180,E1 -11232.544,E2 -11232.544} C_VEL
LIN {X 0,Y 401.275,Z 322.525,A -85,B 0,C 180,E1 -11233.137,E2 -11233.137} C_VEL
LIN {X 0,Y 400.371,Z 334.783,A -85,B 0,C 180,E1 -11233.95,E2 -11233.95} C_VEL
LIN {X 0,Y 399.424,Z 346.383,A -85,B 0,C 180,E1 -11234.958,E2 -11234.958} C_VEL
LIN {X 0,Y 398.634,Z 357.035,A -85,B 0,C 180,E1 -11236.125,E2 -11236.125} C_VEL
LIN {X 0,Y 397.959,Z 365.377,A -85,B 0,C 180,E1 -11237.246,E2 -11237.246} C_VEL
LIN {X 0,Y 397.202,Z 373.261,A -85,B 0,C 180,E1 -11238.518,E2 -11238.518} C_VEL
LIN {X 0,Y 396.605,Z 380.967,A -85,B 0,C 180,E1 -11240.05,E2 -11240.05} C_VEL
LIN {X 0,Y 396.16,Z 388.078,A -85,B 0,C 180,E1 -11241.84,E2 -11241.84} C_VEL
LIN {X 0,Y 395.896,Z 392.811,A -85,B 0,C 180,E1 -11243.374,E2 -11243.374} C_VEL
LIN {X 0,Y 395.829,Z 396.429,A -85,B 0,C 180,E1 -11244.906,E2 -11244.906} C_VEL
LIN {X 0,Y 395.774,Z 398.294,A -85,B 0,C 180,E1 -11245.926,E2 -11245.926} C_VEL
LIN {X 0,Y 395.805,Z 400.695,A -85,B 0,C 180,E1 -11247.964,E2 -11247.964} C_VEL
LIN {X 0,Y 395.812,Z 401.305,A -85,B 0,C 180,E1 -11248.982,E2 -11248.982} C_VEL
LIN {X 0,Y 395.801,Z 401.52,A -85,B 0,C 180,E1 -11249.999,E2 -11249.999} C_VEL
LIN {X 0,Y 395.812,Z 401.302,A -85,B 0,C 180,E1 -11251.017,E2 -11251.017} C_VEL
LIN {X 0,Y 395.804,Z 400.692,A -85,B 0,C 180,E1 -11252.035,E2 -11252.035} C_VEL
LIN {X 0,Y 395.775,Z 398.287,A -85,B 0,C 180,E1 -11254.073,E2 -11254.073} C_VEL
LIN {X 0,Y 395.822,Z 394.882,A -85,B 0,C 180,E1 -11255.799,E2 -11255.799} C_VEL
LIN {X 0,Y 396.061,Z 389.753,A -85,B 0,C 180,E1 -11257.647,E2 -11257.647} C_VEL
LIN {X 0,Y 396.369,Z 384.208,A -85,B 0,C 180,E1 -11259.182,E2 -11259.182} C_VEL
LIN {X 0,Y 396.852,Z 377.29,A -85,B 0,C 180,E1 -11260.716,E2 -11260.716} C_VEL
LIN {X 0,Y 397.64,Z 368.642,A -85,B 0,C 180,E1 -11262.244,E2 -11262.244} C_VEL
LIN {X 0,Y 398.347,Z 359.999,A -85,B 0,C 180,E1 -11263.488,E2 -11263.488} C_VEL
LIN {X 0,Y 399.199,Z 349.337,A -85,B 0,C 180,E1 -11264.737,E2 -11264.737} C_VEL
LIN {X 0,Y 400.096,Z 337.856,A -85,B 0,C 180,E1 -11265.799,E2 -11265.799} C_VEL
LIN {X 0,Y 401.024,Z 325.522,A -85,B 0,C 180,E1 -11266.676,E2 -11266.676} C_VEL
LIN {X 0,Y 401.722,Z 313.846,A -85,B 0,C 180,E1 -11267.301,E2 -11267.301} C_VEL
LIN {X 0,Y 402.363,Z 301.407,A -85,B 0,C 180,E1 -11267.765,E2 -11267.765} C_VEL
LIN {X 0,Y 402.738,Z 285.543,A -85,B 0,C 180,E1 -11268.109,E2 -11268.109} C_VEL
LIN {X 0,Y 403.443,Z 217.491,A -85,B 0,C 180,E1 -11269.327,E2 -11269.327} C_VEL
LIN {X 0,Y 399.251,Z 190.752,A -85,B 0,C 180,E1 -11270.035,E2 -11270.035} C_VEL
LIN {X 0,Y 398.882,Z 188.409,A -85,B 0,C 180,E1 -11270.127,E2 -11270.127} C_VEL
LIN {X 0,Y 400.272,Z 170.337,A -85,B 0,C 180,E1 -11273.817,E2 -11273.817} C_VEL
LIN {X 0,Y 400.376,Z 165.1,A -85,B 0,C 180,E1 -11274.915,E2 -11274.915} C_VEL
LIN {X 0,Y 397.928,Z 152.584,A -85,B 0,C 180,E1 -11277.752,E2 -11277.752} C_VEL
LIN {X 0,Y 397.15,Z 149.016,A -85,B 0,C 180,E1 -11278.612,E2 -11278.612} C_VEL
LIN {X 0,Y 397.074,Z 149.022,A -85,B 0,C 180,E1 -11282.071,E2 -11282.071} C_VEL
LIN {X 0,Y 397.112,Z 149.022,A -85,B 0,C 180,E1 -11285.502,E2 -11285.502} C_VEL
LIN {X 0,Y 397.089,Z 149.02,A -85,B 0,C 180,E1 -11288.854,E2 -11288.854} C_VEL
LIN {X 0,Y 397.052,Z 149.023,A -85,B 0,C 180,E1 -11292.268,E2 -11292.268} C_VEL
LIN {X 0,Y 397.08,Z 149.024,A -85,B 0,C 180,E1 -11295.068,E2 -11295.068} C_VEL
LIN {X 0,Y 397.046,Z 149.024,A -85,B 0,C 180,E1 -11298.023,E2 -11298.023} C_VEL
LIN {X 0,Y 397.087,Z 149.019,A -85,B 0,C 180,E1 -11301.723,E2 -11301.723} C_VEL
LIN {X 0,Y 397.11,Z 149.017,A -85,B 0,C 180,E1 -11305.505,E2 -11305.505} C_VEL
LIN {X 0,Y 397.068,Z 149.024,A -85,B 0,C 180,E1 -11309.117,E2 -11309.117} C_VEL
LIN {X 0,Y 397.07,Z 149.022,A -85,B 0,C 180,E1 -11312.246,E2 -11312.246} C_VEL
LIN {X 0,Y 397.094,Z 149.022,A -85,B 0,C 180,E1 -11314.864,E2 -11314.864} C_VEL
LIN {X 0,Y 397.085,Z 149.021,A -85,B 0,C 180,E1 -11318.181,E2 -11318.181} C_VEL
LIN {X 0,Y 397.1,Z 149.017,A -85,B 0,C 180,E1 -11321.424,E2 -11321.424} C_VEL
LIN {X 0,Y 397.114,Z 149.019,A -85,B 0,C 180,E1 -11324.605,E2 -11324.605} C_VEL
LIN {X 0,Y 397.204,Z 149.005,A -85,B 0,C 180,E1 -11327.741,E2 -11327.741} C_VEL
LIN {X 0,Y 397.217,Z 149.003,A -85,B 0,C 180,E1 -11330.837,E2 -11330.837} C_VEL
LIN {X 0,Y 397.309,Z 148.995,A -85,B 0,C 180,E1 -11333.908,E2 -11333.908} C_VEL
LIN {X 0,Y 397.427,Z 148.982,A -85,B 0,C 180,E1 -11337.973,E2 -11337.973} C_VEL
LIN {X 0,Y 397.429,Z 148.981,A -85,B 0,C 180,E1 -11342.027,E2 -11342.027} C_VEL
LIN {X 0,Y 397.292,Z 148.994,A -85,B 0,C 180,E1 -11346.443,E2 -11346.443} C_VEL
LIN {X 0,Y 397.225,Z 149.003,A -85,B 0,C 180,E1 -11349.163,E2 -11349.163} C_VEL
LIN {X 0,Y 397.209,Z 149.004,A -85,B 0,C 180,E1 -11352.259,E2 -11352.259} C_VEL
LIN {X 0,Y 397.115,Z 149.02,A -85,B 0,C 180,E1 -11355.395,E2 -11355.395} C_VEL
LIN {X 0,Y 397.105,Z 149.016,A -85,B 0,C 180,E1 -11358.576,E2 -11358.576} C_VEL
LIN {X 0,Y 397.098,Z 149.019,A -85,B 0,C 180,E1 -11361.819,E2 -11361.819} C_VEL
LIN {X 0,Y 397.089,Z 149.023,A -85,B 0,C 180,E1 -11365.136,E2 -11365.136} C_VEL
LIN {X 0,Y 397.063,Z 149.022,A -85,B 0,C 180,E1 -11368.548,E2 -11368.548} C_VEL
LIN {X 0,Y 397.073,Z 149.02,A -85,B 0,C 180,E1 -11371.837,E2 -11371.837} C_VEL
LIN {X 0,Y 397.111,Z 149.017,A -85,B 0,C 180,E1 -11374.495,E2 -11374.495} C_VEL
LIN {X 0,Y 397.087,Z 149.019,A -85,B 0,C 180,E1 -11378.277,E2 -11378.277} C_VEL
LIN {X 0,Y 397.048,Z 149.023,A -85,B 0,C 180,E1 -11381.978,E2 -11381.978} C_VEL
LIN {X 0,Y 397.081,Z 149.022,A -85,B 0,C 180,E1 -11385.07,E2 -11385.07} C_VEL
LIN {X 0,Y 397.057,Z 149.023,A -85,B 0,C 180,E1 -11388.023,E2 -11388.023} C_VEL
LIN {X 0,Y 397.096,Z 149.018,A -85,B 0,C 180,E1 -11391.145,E2 -11391.145} C_VEL
LIN {X 0,Y 397.116,Z 149.021,A -85,B 0,C 180,E1 -11394.498,E2 -11394.498} C_VEL
LIN {X 0,Y 397.076,Z 149.022,A -85,B 0,C 180,E1 -11397.929,E2 -11397.929} C_VEL
LIN {X 0,Y 397.116,Z 149.022,A -85,B 0,C 180,E1 -11400.296,E2 -11400.296} C_VEL
LIN {X 0,Y 397.09,Z 149.02,A -85,B 0,C 180,E1 -11403.74,E2 -11403.74} C_VEL
LIN {X 0,Y 397.167,Z 149.166,A -85,B 0,C 180,E1 -11406.872,E2 -11406.872} C_VEL
LIN {X 0,Y 399.407,Z 160.591,A -85,B 0,C 180,E1 -11409.725,E2 -11409.725} C_VEL
LIN {X 0,Y 399.441,Z 161.836,A -85,B 0,C 180,E1 -11409.991,E2 -11409.991} C_VEL
LIN {X 0,Y 403.87,Z 183.093,A -85,B 0,C 180,E1 -11410.617,E2 -11410.617} C_VEL
LIN {X 0,Y 402.818,Z 266.918,A -85,B 0,C 180,E1 -11412.125,E2 -11412.125} C_VEL
LIN {X 0,Y 402.508,Z 279.561,A -85,B 0,C 180,E1 -11412.504,E2 -11412.504} C_VEL
LIN {X 0,Y 401.913,Z 292.402,A -85,B 0,C 180,E1 -11413.1,E2 -11413.1} C_VEL
LIN {X 0,Y 401.204,Z 304.264,A -85,B 0,C 180,E1 -11413.855,E2 -11413.855} C_VEL
LIN {X 0,Y 400.504,Z 315.017,A -85,B 0,C 180,E1 -11414.74,E2 -11414.74} C_VEL
LIN {X 0,Y 399.773,Z 325.971,A -85,B 0,C 180,E1 -11415.883,E2 -11415.883} C_VEL
LIN {X 0,Y 398.897,Z 334.869,A -85,B 0,C 180,E1 -11417.019,E2 -11417.019} C_VEL
LIN {X 0,Y 398.064,Z 344.502,A -85,B 0,C 180,E1 -11418.544,E2 -11418.544} C_VEL
LIN {X 0,Y 397.358,Z 352.186,A -85,B 0,C 180,E1 -11420.071,E2 -11420.071} C_VEL
LIN {X 0,Y 396.713,Z 359.236,A -85,B 0,C 180,E1 -11421.853,E2 -11421.853} C_VEL
LIN {X 0,Y 396.422,Z 364.103,A -85,B 0,C 180,E1 -11423.447,E2 -11423.447} C_VEL
LIN {X 0,Y 396.102,Z 367.522,A -85,B 0,C 180,E1 -11424.911,E2 -11424.911} C_VEL
LIN {X 0,Y 395.985,Z 369.378,A -85,B 0,C 180,E1 -11425.93,E2 -11425.93} C_VEL
LIN {X 0,Y 395.974,Z 370.773,A -85,B 0,C 180,E1 -11426.948,E2 -11426.948} C_VEL
LIN {X 0,Y 395.832,Z 372.198,A -85,B 0,C 180,E1 -11428.68,E2 -11428.68} C_VEL
LIN {X 0,Y 395.803,Z 372.615,A -85,B 0,C 180,E1 -11430.001,E2 -11430.001} C_VEL
LIN {X 0,Y 395.905,Z 371.841,A -85,B 0,C 180,E1 -11432.035,E2 -11432.035} C_VEL
LIN {X 0,Y 395.968,Z 370.815,A -85,B 0,C 180,E1 -11433.1,E2 -11433.1} C_VEL
LIN {X 0,Y 395.305,Z 369.759,A -85,B 0,C 180,E1 -11433.935,E2 -11433.935} C_VEL
LIN {X 0,Y 392.585,Z 367.539,A -85,B 0,C 180,E1 -11435.288,E2 -11435.288} C_VEL
LIN {X 0,Y 390.35,Z 365.344,A -85,B 0,C 180,E1 -11436.361,E2 -11436.361} C_VEL
LIN {X 0,Y 389.456,Z 363.29,A -85,B 0,C 180,E1 -11437.168,E2 -11437.168} C_VEL
LIN {X 0,Y 389.416,Z 362.517,A -85,B 0,C 180,E1 -11437.436,E2 -11437.436} C_VEL
LIN {X 0,Y 389.804,Z 358.042,A -85,B 0,C 180,E1 -11438.816,E2 -11438.816} C_VEL
LIN {X 0,Y 390.471,Z 351.736,A -85,B 0,C 180,E1 -11440.369,E2 -11440.369} C_VEL
LIN {X 0,Y 391.197,Z 343.845,A -85,B 0,C 180,E1 -11441.924,E2 -11441.924} C_VEL
LIN {X 0,Y 391.958,Z 335.797,A -85,B 0,C 180,E1 -11443.216,E2 -11443.216} C_VEL
LIN {X 0,Y 392.95,Z 325.97,A -85,B 0,C 180,E1 -11444.501,E2 -11444.501} C_VEL
LIN {X 0,Y 393.627,Z 316.306,A -85,B 0,C 180,E1 -11445.535,E2 -11445.535} C_VEL
LIN {X 0,Y 394.387,Z 305.842,A -85,B 0,C 180,E1 -11446.433,E2 -11446.433} C_VEL
LIN {X 0,Y 395.104,Z 294.361,A -85,B 0,C 180,E1 -11447.201,E2 -11447.201} C_VEL
LIN {X 0,Y 395.733,Z 281.373,A -85,B 0,C 180,E1 -11447.84,E2 -11447.84} C_VEL
LIN {X 0,Y 396.187,Z 268.644,A -85,B 0,C 180,E1 -11448.253,E2 -11448.253} C_VEL
LIN {X 0,Y 397.192,Z 183.939,A -85,B 0,C 180,E1 -11449.813,E2 -11449.813} C_VEL
LIN {X 0,Y 392.734,Z 163.26,A -85,B 0,C 180,E1 -11450.446,E2 -11450.446} C_VEL
LIN {X 0,Y 392.405,Z 161.761,A -85,B 0,C 180,E1 -11450.541,E2 -11450.541} C_VEL
LIN {X 0,Y 390.105,Z 149.891,A -85,B 0,C 180,E1 -11453.561,E2 -11453.561} C_VEL
LIN {X 0,Y 390.057,Z 149.897,A -85,B 0,C 180,E1 -11456.773,E2 -11456.773} C_VEL
LIN {X 0,Y 390.039,Z 149.898,A -85,B 0,C 180,E1 -11460.3,E2 -11460.3} C_VEL
LIN {X 0,Y 390.07,Z 149.895,A -85,B 0,C 180,E1 -11464.024,E2 -11464.024} C_VEL
LIN {X 0,Y 390.041,Z 149.903,A -85,B 0,C 180,E1 -11467.55,E2 -11467.55} C_VEL
LIN {X 0,Y 390.02,Z 149.9,A -85,B 0,C 180,E1 -11470.815,E2 -11470.815} C_VEL
LIN {X 0,Y 390.054,Z 149.896,A -85,B 0,C 180,E1 -11473.886,E2 -11473.886} C_VEL
LIN {X 0,Y 390.055,Z 149.896,A -85,B 0,C 180,E1 -11476.789,E2 -11476.789} C_VEL
LIN {X 0,Y 390.011,Z 149.903,A -85,B 0,C 180,E1 -11479.555,E2 -11479.555} C_VEL
LIN {X 0,Y 390.04,Z 149.897,A -85,B 0,C 180,E1 -11482.45,E2 -11482.45} C_VEL
LIN {X 0,Y 390.061,Z 149.894,A -85,B 0,C 180,E1 -11486.044,E2 -11486.044} C_VEL
LIN {X 0,Y 390.042,Z 149.896,A -85,B 0,C 180,E1 -11489.87,E2 -11489.87} C_VEL
LIN {X 0,Y 390.047,Z 149.898,A -85,B 0,C 180,E1 -11493.227,E2 -11493.227} C_VEL
LIN {X 0,Y 390.067,Z 149.899,A -85,B 0,C 180,E1 -11496.763,E2 -11496.763} C_VEL
LIN {X 0,Y 390.101,Z 149.889,A -85,B 0,C 180,E1 -11499.983,E2 -11499.983} C_VEL
LIN {X 0,Y 390.104,Z 149.889,A -85,B 0,C 180,E1 -11503.247,E2 -11503.247} C_VEL
LIN {X 0,Y 390.193,Z 149.883,A -85,B 0,C 180,E1 -11506.561,E2 -11506.561} C_VEL
LIN {X 0,Y 390.163,Z 149.881,A -85,B 0,C 180,E1 -11509.623,E2 -11509.623} C_VEL
LIN {X 0,Y 390.243,Z 149.873,A -85,B 0,C 180,E1 -11512.758,E2 -11512.758} C_VEL
LIN {X 0,Y 390.195,Z 149.878,A -85,B 0,C 180,E1 -11514.833,E2 -11514.833} C_VEL
LIN {X 0,Y 390.403,Z 149.855,A -85,B 0,C 180,E1 -11517.937,E2 -11517.937} C_VEL
LIN {X 0,Y 390.4,Z 149.858,A -85,B 0,C 180,E1 -11522.063,E2 -11522.063} C_VEL
LIN {X 0,Y 390.271,Z 149.871,A -85,B 0,C 180,E1 -11526.203,E2 -11526.203} C_VEL
LIN {X 0,Y 390.181,Z 149.88,A -85,B 0,C 180,E1 -11529.329,E2 -11529.329} C_VEL
LIN {X 0,Y 390.15,Z 149.883,A -85,B 0,C 180,E1 -11532.484,E2 -11532.484} C_VEL
LIN {X 0,Y 390.05,Z 149.901,A -85,B 0,C 180,E1 -11535.681,E2 -11535.681} C_VEL
LIN {X 0,Y 390.041,Z 149.897,A -85,B 0,C 180,E1 -11538.925,E2 -11538.925} C_VEL
LIN {X 0,Y 390.029,Z 149.898,A -85,B 0,C 180,E1 -11542.235,E2 -11542.235} C_VEL
LIN {X 0,Y 390.048,Z 149.898,A -85,B 0,C 180,E1 -11545.722,E2 -11545.722} C_VEL
LIN {X 0,Y 390.02,Z 149.904,A -85,B 0,C 180,E1 -11549.113,E2 -11549.113} C_VEL
LIN {X 0,Y 390.038,Z 149.899,A -85,B 0,C 180,E1 -11552.722,E2 -11552.722} C_VEL
LIN {X 0,Y 390.042,Z 149.896,A -85,B 0,C 180,E1 -11555.823,E2 -11555.823} C_VEL
LIN {X 0,Y 390.038,Z 149.9,A -85,B 0,C 180,E1 -11559.213,E2 -11559.213} C_VEL
LIN {X 0,Y 390.029,Z 149.899,A -85,B 0,C 180,E1 -11562.372,E2 -11562.372} C_VEL
LIN {X 0,Y 390.04,Z 149.897,A -85,B 0,C 180,E1 -11565.354,E2 -11565.354} C_VEL
LIN {X 0,Y 390.015,Z 149.901,A -85,B 0,C 180,E1 -11568.185,E2 -11568.185} C_VEL
LIN {X 0,Y 390.058,Z 149.898,A -85,B 0,C 180,E1 -11570.904,E2 -11570.904} C_VEL
LIN {X 0,Y 390.082,Z 149.895,A -85,B 0,C 180,E1 -11574.793,E2 -11574.793} C_VEL
LIN {X 0,Y 390.024,Z 149.904,A -85,B 0,C 180,E1 -11578.496,E2 -11578.496} C_VEL
LIN {X 0,Y 390.114,Z 150.014,A -85,B 0,C 180,E1 -11581.122,E2 -11581.122} C_VEL
LIN {X 0,Y 392.678,Z 162.484,A -85,B 0,C 180,E1 -11584.047,E2 -11584.047} C_VEL
LIN {X 0,Y 393.555,Z 167.512,A -85,B 0,C 180,E1 -11585.187,E2 -11585.187} C_VEL
LIN {X 0,Y 392.548,Z 180.547,A -85,B 0,C 180,E1 -11587.915,E2 -11587.915} C_VEL
LIN {X 0,Y 391.997,Z 188.272,A -85,B 0,C 180,E1 -11589.52,E2 -11589.52} C_VEL
LIN {X 0,Y 396.497,Z 216.399,A -85,B 0,C 180,E1 -11590.294,E2 -11590.294} C_VEL
LIN {X 0,Y 396.863,Z 221.262,A -85,B 0,C 180,E1 -11590.404,E2 -11590.404} C_VEL
LIN {X 0,Y 395.803,Z 296.901,A -85,B 0,C 180,E1 -11591.796,E2 -11591.796} C_VEL
LIN {X 0,Y 395.199,Z 310.128,A -85,B 0,C 180,E1 -11592.236,E2 -11592.236} C_VEL
LIN {X 0,Y 394.484,Z 322.272,A -85,B 0,C 180,E1 -11592.838,E2 -11592.838} C_VEL
LIN {X 0,Y 393.552,Z 334.528,A -85,B 0,C 180,E1 -11593.664,E2 -11593.664} C_VEL
LIN {X 0,Y 392.546,Z 346.123,A -85,B 0,C 180,E1 -11594.687,E2 -11594.687} C_VEL
LIN {X 0,Y 391.769,Z 356.151,A -85,B 0,C 180,E1 -11595.8,E2 -11595.8} C_VEL
LIN {X 0,Y 391.006,Z 365.119,A -85,B 0,C 180,E1 -11597.016,E2 -11597.016} C_VEL
LIN {X 0,Y 390.23,Z 373.003,A -85,B 0,C 180,E1 -11598.31,E2 -11598.31} C_VEL
LIN {X 0,Y 389.591,Z 380.708,A -85,B 0,C 180,E1 -11599.869,E2 -11599.869} C_VEL
LIN {X 0,Y 389.105,Z 387.819,A -85,B 0,C 180,E1 -11601.692,E2 -11601.692} C_VEL
LIN {X 0,Y 388.826,Z 392.55,A -85,B 0,C 180,E1 -11603.252,E2 -11603.252} C_VEL
LIN {X 0,Y 388.724,Z 396.169,A -85,B 0,C 180,E1 -11604.813,E2 -11604.813} C_VEL
LIN {X 0,Y 388.698,Z 398.036,A -85,B 0,C 180,E1 -11605.852,E2 -11605.852} C_VEL
LIN {X 0,Y 388.702,Z 400.436,A -85,B 0,C 180,E1 -11607.927,E2 -11607.927} C_VEL
LIN {X 0,Y 388.741,Z 401.047,A -85,B 0,C 180,E1 -11608.964,E2 -11608.964} C_VEL
LIN {X 0,Y 388.729,Z 401.262,A -85,B 0,C 180,E1 -11609.999,E2 -11609.999} C_VEL
LIN {X 0,Y 388.741,Z 401.044,A -85,B 0,C 180,E1 -11611.035,E2 -11611.035} C_VEL
LIN {X 0,Y 388.702,Z 400.432,A -85,B 0,C 180,E1 -11612.072,E2 -11612.072} C_VEL
LIN {X 0,Y 388.699,Z 398.028,A -85,B 0,C 180,E1 -11614.147,E2 -11614.147} C_VEL
LIN {X 0,Y 388.773,Z 394.048,A -85,B 0,C 180,E1 -11616.142,E2 -11616.142} C_VEL
LIN {X 0,Y 388.994,Z 389.492,A -85,B 0,C 180,E1 -11617.787,E2 -11617.787} C_VEL
LIN {X 0,Y 389.338,Z 383.946,A -85,B 0,C 180,E1 -11619.349,E2 -11619.349} C_VEL
LIN {X 0,Y 389.84,Z 377.027,A -85,B 0,C 180,E1 -11620.911,E2 -11620.911} C_VEL
LIN {X 0,Y 390.685,Z 368.38,A -85,B 0,C 180,E1 -11622.466,E2 -11622.466} C_VEL
LIN {X 0,Y 391.585,Z 358.366,A -85,B 0,C 180,E1 -11623.911,E2 -11623.911} C_VEL
LIN {X 0,Y 392.35,Z 348.6,A -85,B 0,C 180,E1 -11625.053,E2 -11625.053} C_VEL
LIN {X 0,Y 393.26,Z 337.592,A -85,B 0,C 180,E1 -11626.081,E2 -11626.081} C_VEL
LIN {X 0,Y 394.217,Z 325.257,A -85,B 0,C 180,E1 -11626.973,E2 -11626.973} C_VEL
LIN {X 0,Y 394.958,Z 313.579,A -85,B 0,C 180,E1 -11627.607,E2 -11627.607} C_VEL
LIN {X 0,Y 395.607,Z 301.135,A -85,B 0,C 180,E1 -11628.079,E2 -11628.079} C_VEL
LIN {X 0,Y 395.996,Z 285.264,A -85,B 0,C 180,E1 -11628.428,E2 -11628.428} C_VEL
LIN {X 0,Y 396.737,Z 218.109,A -85,B 0,C 180,E1 -11629.651,E2 -11629.651} C_VEL
LIN {X 0,Y 391.998,Z 188.373,A -85,B 0,C 180,E1 -11630.462,E2 -11630.462} C_VEL
LIN {X 0,Y 393.468,Z 170.072,A -85,B 0,C 180,E1 -11634.255,E2 -11634.255} C_VEL
LIN {X 0,Y 393.371,Z 166.139,A -85,B 0,C 180,E1 -11635.106,E2 -11635.106} C_VEL
LIN {X 0,Y 391.056,Z 154.237,A -85,B 0,C 180,E1 -11637.856,E2 -11637.856} C_VEL
LIN {X 0,Y 390.097,Z 149.894,A -85,B 0,C 180,E1 -11638.91,E2 -11638.91} C_VEL
LIN {X 0,Y 390.038,Z 149.897,A -85,B 0,C 180,E1 -11642.721,E2 -11642.721} C_VEL
LIN {X 0,Y 390.05,Z 149.898,A -85,B 0,C 180,E1 -11645.824,E2 -11645.824} C_VEL
LIN {X 0,Y 390.033,Z 149.902,A -85,B 0,C 180,E1 -11649.211,E2 -11649.211} C_VEL
LIN {X 0,Y 390.027,Z 149.898,A -85,B 0,C 180,E1 -11652.371,E2 -11652.371} C_VEL
LIN {X 0,Y 390.035,Z 149.902,A -85,B 0,C 180,E1 -11655.353,E2 -11655.353} C_VEL
LIN {X 0,Y 390.009,Z 149.9,A -85,B 0,C 180,E1 -11658.184,E2 -11658.184} C_VEL
LIN {X 0,Y 390.053,Z 149.9,A -85,B 0,C 180,E1 -11660.903,E2 -11660.903} C_VEL
LIN {X 0,Y 390.062,Z 149.898,A -85,B 0,C 180,E1 -11664.791,E2 -11664.791} C_VEL
LIN {X 0,Y 390.014,Z 149.902,A -85,B 0,C 180,E1 -11668.495,E2 -11668.495} C_VEL
LIN {X 0,Y 390.017,Z 149.9,A -85,B 0,C 180,E1 -11672.062,E2 -11672.062} C_VEL
LIN {X 0,Y 390.033,Z 149.897,A -85,B 0,C 180,E1 -11675.516,E2 -11675.516} C_VEL
LIN {X 0,Y 390.043,Z 149.899,A -85,B 0,C 180,E1 -11678.877,E2 -11678.877} C_VEL
LIN {X 0,Y 390.097,Z 149.893,A -85,B 0,C 180,E1 -11682.712,E2 -11682.712} C_VEL
LIN {X 0,Y 390.186,Z 149.882,A -85,B 0,C 180,E1 -11686.561,E2 -11686.561} C_VEL
LIN {X 0,Y 390.175,Z 149.882,A -85,B 0,C 180,E1 -11690.671,E2 -11690.671} C_VEL
LIN {X 0,Y 390.264,Z 149.871,A -85,B 0,C 180,E1 -11693.797,E2 -11693.797} C_VEL
LIN {X 0,Y 390.393,Z 149.858,A -85,B 0,C 180,E1 -11697.937,E2 -11697.937} C_VEL
LIN {X 0,Y 390.396,Z 149.857,A -85,B 0,C 180,E1 -11702.063,E2 -11702.063} C_VEL
LIN {X 0,Y 390.254,Z 149.87,A -85,B 0,C 180,E1 -11706.432,E2 -11706.432} C_VEL
LIN {X 0,Y 390.183,Z 149.881,A -85,B 0,C 180,E1 -11709.329,E2 -11709.329} C_VEL
LIN {X 0,Y 390.161,Z 149.881,A -85,B 0,C 180,E1 -11712.484,E2 -11712.484} C_VEL
LIN {X 0,Y 390.058,Z 149.899,A -85,B 0,C 180,E1 -11715.68,E2 -11715.68} C_VEL
LIN {X 0,Y 390.067,Z 149.895,A -85,B 0,C 180,E1 -11718.924,E2 -11718.924} C_VEL
LIN {X 0,Y 390.033,Z 149.897,A -85,B 0,C 180,E1 -11722.235,E2 -11722.235} C_VEL
LIN {X 0,Y 390.042,Z 149.898,A -85,B 0,C 180,E1 -11725.723,E2 -11725.723} C_VEL
LIN {X 0,Y 390.022,Z 149.905,A -85,B 0,C 180,E1 -11729.113,E2 -11729.113} C_VEL
LIN {X 0,Y 390.034,Z 149.9,A -85,B 0,C 180,E1 -11732.723,E2 -11732.723} C_VEL
LIN {X 0,Y 390.037,Z 149.897,A -85,B 0,C 180,E1 -11735.823,E2 -11735.823} C_VEL
LIN {X 0,Y 390.032,Z 149.9,A -85,B 0,C 180,E1 -11739.213,E2 -11739.213} C_VEL
LIN {X 0,Y 390.026,Z 149.9,A -85,B 0,C 180,E1 -11742.373,E2 -11742.373} C_VEL
LIN {X 0,Y 390.039,Z 149.897,A -85,B 0,C 180,E1 -11745.355,E2 -11745.355} C_VEL
LIN {X 0,Y 390.02,Z 149.901,A -85,B 0,C 180,E1 -11748.187,E2 -11748.187} C_VEL
LIN {X 0,Y 390.059,Z 149.897,A -85,B 0,C 180,E1 -11750.905,E2 -11750.905} C_VEL
LIN {X 0,Y 390.082,Z 149.894,A -85,B 0,C 180,E1 -11754.794,E2 -11754.794} C_VEL
LIN {X 0,Y 390.022,Z 149.903,A -85,B 0,C 180,E1 -11758.497,E2 -11758.497} C_VEL
LIN {X 0,Y 390.034,Z 149.902,A -85,B 0,C 180,E1 -11762.065,E2 -11762.065} C_VEL
LIN {X 0,Y 390.051,Z 149.896,A -85,B 0,C 180,E1 -11765.518,E2 -11765.518} C_VEL
LIN {X 0,Y 390.121,Z 150.021,A -85,B 0,C 180,E1 -11766.582,E2 -11766.582} C_VEL
LIN {X 0,Y 392.475,Z 161.908,A -85,B 0,C 180,E1 -11769.601,E2 -11769.601} C_VEL
LIN {X 0,Y 396.832,Z 182.192,A -85,B 0,C 180,E1 -11770.237,E2 -11770.237} C_VEL
LIN {X 0,Y 397.257,Z 184.3,A -85,B 0,C 180,E1 -11770.299,E2 -11770.299} C_VEL
LIN {X 0,Y 396.071,Z 267.199,A -85,B 0,C 180,E1 -11771.81,E2 -11771.81} C_VEL
LIN {X 0,Y 395.751,Z 279.832,A -85,B 0,C 180,E1 -11772.196,E2 -11772.196} C_VEL
LIN {X 0,Y 395.151,Z 292.669,A -85,B 0,C 180,E1 -11772.802,E2 -11772.802} C_VEL
LIN {X 0,Y 394.412,Z 304.529,A -85,B 0,C 180,E1 -11773.569,E2 -11773.569} C_VEL
LIN {X 0,Y 393.677,Z 315.281,A -85,B 0,C 180,E1 -11774.468,E2 -11774.468} C_VEL
LIN {X 0,Y 392.908,Z 326.233,A -85,B 0,C 180,E1 -11775.631,E2 -11775.631} C_VEL
LIN {X 0,Y 391.993,Z 335.131,A -85,B 0,C 180,E1 -11776.786,E2 -11776.786} C_VEL
LIN {X 0,Y 391.284,Z 343.286,A -85,B 0,C 180,E1 -11778.08,E2 -11778.08} C_VEL
LIN {X 0,Y 390.5,Z 351.276,A -85,B 0,C 180,E1 -11779.632,E2 -11779.632} C_VEL
LIN {X 0,Y 389.861,Z 357.69,A -85,B 0,C 180,E1 -11781.187,E2 -11781.187} C_VEL
LIN {X 0,Y 389.381,Z 363.683,A -85,B 0,C 180,E1 -11783.077,E2 -11783.077} C_VEL
LIN {X 0,Y 389.052,Z 367.781,A -85,B 0,C 180,E1 -11784.818,E2 -11784.818} C_VEL
LIN {X 0,Y 388.905,Z 369.638,A -85,B 0,C 180,E1 -11785.855,E2 -11785.855} C_VEL
LIN {X 0,Y 388.88,Z 371.033,A -85,B 0,C 180,E1 -11786.893,E2 -11786.893} C_VEL
LIN {X 0,Y 388.823,Z 372.026,A -85,B 0,C 180,E1 -11787.929,E2 -11787.929} C_VEL
LIN {X 0,Y 388.731,Z 372.873,A -85,B 0,C 180,E1 -11790.001,E2 -11790.001} C_VEL
LIN {X 0,Y 388.75,Z 372.684,A -85,B 0,C 180,E1 -11791.036,E2 -11791.036} C_VEL
LIN {X 0,Y 388.823,Z 372.1,A -85,B 0,C 180,E1 -11792.072,E2 -11792.072} C_VEL
LIN {X 0,Y 388.876,Z 371.135,A -85,B 0,C 180,E1 -11793.108,E2 -11793.108} C_VEL
LIN {X 0,Y 388.894,Z 369.785,A -85,B 0,C 180,E1 -11794.146,E2 -11794.146} C_VEL
LIN {X 0,Y 389.174,Z 366.923,A -85,B 0,C 180,E1 -11795.701,E2 -11795.701} C_VEL
LIN {X 0,Y 389.416,Z 362.517,A -85,B 0,C 180,E1 -11797.436,E2 -11797.436} C_VEL
LIN {X 0,Y 388.91,Z 360.15,A -85,B 0,C 180,E1 -11798.23,E2 -11798.23} C_VEL
LIN {X 0,Y 386.446,Z 355.889,A -85,B 0,C 180,E1 -11799.51,E2 -11799.51} C_VEL
LIN {X 0,Y 384.136,Z 351.047,A -85,B 0,C 180,E1 -11800.751,E2 -11800.751} C_VEL
LIN {X 0,Y 383.868,Z 347.656,A -85,B 0,C 180,E1 -11801.472,E2 -11801.472} C_VEL
LIN {X 0,Y 384.714,Z 339.461,A -85,B 0,C 180,E1 -11802.932,E2 -11802.932} C_VEL
LIN {X 0,Y 385.642,Z 330.424,A -85,B 0,C 180,E1 -11804.243,E2 -11804.243} C_VEL
LIN {X 0,Y 386.495,Z 319.938,A -85,B 0,C 180,E1 -11805.474,E2 -11805.474} C_VEL
LIN {X 0,Y 387.341,Z 309.286,A -85,B 0,C 180,E1 -11806.47,E2 -11806.47} C_VEL
LIN {X 0,Y 388.218,Z 296.783,A -85,B 0,C 180,E1 -11807.38,E2 -11807.38} C_VEL
LIN {X 0,Y 388.908,Z 284.662,A -85,B 0,C 180,E1 -11808.027,E2 -11808.027} C_VEL
LIN {X 0,Y 389.339,Z 272.35,A -85,B 0,C 180,E1 -11808.483,E2 -11808.483} C_VEL
LIN {X 0,Y 389.746,Z 252.032,A -85,B 0,C 180,E1 -11808.906,E2 -11808.906} C_VEL
LIN {X 0,Y 390.577,Z 185.217,A -85,B 0,C 180,E1 -11810.143,E2 -11810.143} C_VEL
LIN {X 0,Y 386.15,Z 164.743,A -85,B 0,C 180,E1 -11810.786,E2 -11810.786} C_VEL
LIN {X 0,Y 385.319,Z 162.135,A -85,B 0,C 180,E1 -11810.909,E2 -11810.909} C_VEL
LIN {X 0,Y 383.066,Z 150.771,A -85,B 0,C 180,E1 -11813.877,E2 -11813.877} C_VEL
LIN {X 0,Y 382.996,Z 150.776,A -85,B 0,C 180,E1 -11817.307,E2 -11817.307} C_VEL
LIN {X 0,Y 382.984,Z 150.775,A -85,B 0,C 180,E1 -11820.919,E2 -11820.919} C_VEL
LIN {X 0,Y 383.02,Z 150.771,A -85,B 0,C 180,E1 -11824.668,E2 -11824.668} C_VEL
LIN {X 0,Y 382.995,Z 150.777,A -85,B 0,C 180,E1 -11827.902,E2 -11827.902} C_VEL
LIN {X 0,Y 382.964,Z 150.783,A -85,B 0,C 180,E1 -11831.35,E2 -11831.35} C_VEL
LIN {X 0,Y 382.996,Z 150.774,A -85,B 0,C 180,E1 -11834.303,E2 -11834.303} C_VEL
LIN {X 0,Y 383.011,Z 150.778,A -85,B 0,C 180,E1 -11837.24,E2 -11837.24} C_VEL
LIN {X 0,Y 382.986,Z 150.775,A -85,B 0,C 180,E1 -11840.419,E2 -11840.419} C_VEL
LIN {X 0,Y 383.014,Z 150.772,A -85,B 0,C 180,E1 -11844.043,E2 -11844.043} C_VEL
LIN {X 0,Y 382.984,Z 150.776,A -85,B 0,C 180,E1 -11847.578,E2 -11847.578} C_VEL
LIN {X 0,Y 382.977,Z 150.777,A -85,B 0,C 180,E1 -11850.299,E2 -11850.299} C_VEL
LIN {X 0,Y 383.003,Z 150.773,A -85,B 0,C 180,E1 -11854.044,E2 -11854.044} C_VEL
LIN {X 0,Y 382.991,Z 150.775,A -85,B 0,C 180,E1 -11857.334,E2 -11857.334} C_VEL
LIN {X 0,Y 383.04,Z 150.774,A -85,B 0,C 180,E1 -11860.715,E2 -11860.715} C_VEL
LIN {X 0,Y 383.017,Z 150.773,A -85,B 0,C 180,E1 -11864.024,E2 -11864.024} C_VEL
LIN {X 0,Y 383.134,Z 150.757,A -85,B 0,C 180,E1 -11867.284,E2 -11867.284} C_VEL
LIN {X 0,Y 383.14,Z 150.761,A -85,B 0,C 180,E1 -11870.498,E2 -11870.498} C_VEL
LIN {X 0,Y 383.23,Z 150.746,A -85,B 0,C 180,E1 -11873.683,E2 -11873.683} C_VEL
LIN {X 0,Y 383.369,Z 150.731,A -85,B 0,C 180,E1 -11877.899,E2 -11877.899} C_VEL
LIN {X 0,Y 383.365,Z 150.734,A -85,B 0,C 180,E1 -11882.101,E2 -11882.101} C_VEL
LIN {X 0,Y 383.229,Z 150.747,A -85,B 0,C 180,E1 -11886.317,E2 -11886.317} C_VEL
LIN {X 0,Y 383.171,Z 150.753,A -85,B 0,C 180,E1 -11888.438,E2 -11888.438} C_VEL
LIN {X 0,Y 383.079,Z 150.769,A -85,B 0,C 180,E1 -11891.643,E2 -11891.643} C_VEL
LIN {X 0,Y 383.05,Z 150.772,A -85,B 0,C 180,E1 -11893.799,E2 -11893.799} C_VEL
LIN {X 0,Y 383.021,Z 150.775,A -85,B 0,C 180,E1 -11897.42,E2 -11897.42} C_VEL
LIN {X 0,Y 383.011,Z 150.772,A -85,B 0,C 180,E1 -11900.64,E2 -11900.64} C_VEL
LIN {X 0,Y 383.005,Z 150.775,A -85,B 0,C 180,E1 -11903.809,E2 -11903.809} C_VEL
LIN {X 0,Y 382.965,Z 150.784,A -85,B 0,C 180,E1 -11907.309,E2 -11907.309} C_VEL
LIN {X 0,Y 382.977,Z 150.78,A -85,B 0,C 180,E1 -11910.919,E2 -11910.919} C_VEL
LIN {X 0,Y 383.01,Z 150.774,A -85,B 0,C 180,E1 -11914.669,E2 -11914.669} C_VEL
LIN {X 0,Y 382.993,Z 150.774,A -85,B 0,C 180,E1 -11917.903,E2 -11917.903} C_VEL
LIN {X 0,Y 382.96,Z 150.78,A -85,B 0,C 180,E1 -11921.351,E2 -11921.351} C_VEL
LIN {X 0,Y 382.988,Z 150.776,A -85,B 0,C 180,E1 -11924.302,E2 -11924.302} C_VEL
LIN {X 0,Y 382.981,Z 150.777,A -85,B 0,C 180,E1 -11927.236,E2 -11927.236} C_VEL
LIN {X 0,Y 382.986,Z 150.779,A -85,B 0,C 180,E1 -11930.419,E2 -11930.419} C_VEL
LIN {X 0,Y 383.023,Z 150.772,A -85,B 0,C 180,E1 -11934.044,E2 -11934.044} C_VEL
LIN {X 0,Y 382.986,Z 150.775,A -85,B 0,C 180,E1 -11937.578,E2 -11937.578} C_VEL
LIN {X 0,Y 383.065,Z 150.868,A -85,B 0,C 180,E1 -11940.797,E2 -11940.797} C_VEL
LIN {X 0,Y 385.59,Z 163.031,A -85,B 0,C 180,E1 -11943.715,E2 -11943.715} C_VEL
LIN {X 0,Y 386.589,Z 168.551,A -85,B 0,C 180,E1 -11944.996,E2 -11944.996} C_VEL
LIN {X 0,Y 386.081,Z 176.379,A -85,B 0,C 180,E1 -11946.676,E2 -11946.676} C_VEL
LIN {X 0,Y 385.112,Z 187.991,A -85,B 0,C 180,E1 -11949.134,E2 -11949.134} C_VEL
LIN {X 0,Y 389.964,Z 218.308,A -85,B 0,C 180,E1 -11949.991,E2 -11949.991} C_VEL
LIN {X 0,Y 390.109,Z 224.88,A -85,B 0,C 180,E1 -11950.124,E2 -11950.124} C_VEL
LIN {X 0,Y 389.056,Z 296.654,A -85,B 0,C 180,E1 -11951.469,E2 -11951.469} C_VEL
LIN {X 0,Y 388.454,Z 309.878,A -85,B 0,C 180,E1 -11951.917,E2 -11951.917} C_VEL
LIN {X 0,Y 387.68,Z 322.018,A -85,B 0,C 180,E1 -11952.527,E2 -11952.527} C_VEL
LIN {X 0,Y 386.72,Z 334.272,A -85,B 0,C 180,E1 -11953.367,E2 -11953.367} C_VEL
LIN {X 0,Y 385.687,Z 345.867,A -85,B 0,C 180,E1 -11954.408,E2 -11954.408} C_VEL
LIN {X 0,Y 384.792,Z 356.715,A -85,B 0,C 180,E1 -11955.64,E2 -11955.64} C_VEL
LIN {X 0,Y 384.045,Z 364.861,A -85,B 0,C 180,E1 -11956.776,E2 -11956.776} C_VEL
LIN {X 0,Y 383.267,Z 372.745,A -85,B 0,C 180,E1 -11958.094,E2 -11958.094} C_VEL
LIN {X 0,Y 382.571,Z 380.45,A -85,B 0,C 180,E1 -11959.682,E2 -11959.682} C_VEL
LIN {X 0,Y 382.04,Z 387.559,A -85,B 0,C 180,E1 -11961.537,E2 -11961.537} C_VEL
LIN {X 0,Y 381.746,Z 392.291,A -85,B 0,C 180,E1 -11963.127,E2 -11963.127} C_VEL
LIN {X 0,Y 381.627,Z 395.909,A -85,B 0,C 180,E1 -11964.716,E2 -11964.716} C_VEL
LIN {X 0,Y 381.622,Z 397.777,A -85,B 0,C 180,E1 -11965.775,E2 -11965.775} C_VEL
LIN {X 0,Y 381.6,Z 400.177,A -85,B 0,C 180,E1 -11967.889,E2 -11967.889} C_VEL
LIN {X 0,Y 381.654,Z 400.788,A -85,B 0,C 180,E1 -11968.944,E2 -11968.944} C_VEL
LIN {X 0,Y 381.66,Z 401.004,A -85,B 0,C 180,E1 -11969.999,E2 -11969.999} C_VEL
LIN {X 0,Y 381.654,Z 400.785,A -85,B 0,C 180,E1 -11971.055,E2 -11971.055} C_VEL
LIN {X 0,Y 381.6,Z 400.172,A -85,B 0,C 180,E1 -11972.11,E2 -11972.11} C_VEL
LIN {X 0,Y 381.624,Z 397.768,A -85,B 0,C 180,E1 -11974.224,E2 -11974.224} C_VEL
LIN {X 0,Y 381.685,Z 394.122,A -85,B 0,C 180,E1 -11976.115,E2 -11976.115} C_VEL
LIN {X 0,Y 381.921,Z 389.23,A -85,B 0,C 180,E1 -11977.932,E2 -11977.932} C_VEL
LIN {X 0,Y 382.301,Z 383.685,A -85,B 0,C 180,E1 -11979.523,E2 -11979.523} C_VEL
LIN {X 0,Y 382.844,Z 376.765,A -85,B 0,C 180,E1 -11981.113,E2 -11981.113} C_VEL
LIN {X 0,Y 383.721,Z 368.117,A -85,B 0,C 180,E1 -11982.696,E2 -11982.696} C_VEL
LIN {X 0,Y 384.641,Z 358.485,A -85,B 0,C 180,E1 -11984.115,E2 -11984.115} C_VEL
LIN {X 0,Y 385.472,Z 348.337,A -85,B 0,C 180,E1 -11985.329,E2 -11985.329} C_VEL
LIN {X 0,Y 386.446,Z 337.328,A -85,B 0,C 180,E1 -11986.372,E2 -11986.372} C_VEL
LIN {X 0,Y 387.419,Z 324.992,A -85,B 0,C 180,E1 -11987.28,E2 -11987.28} C_VEL
LIN {X 0,Y 388.205,Z 313.313,A -85,B 0,C 180,E1 -11987.924,E2 -11987.924} C_VEL
LIN {X 0,Y 388.87,Z 300.864,A -85,B 0,C 180,E1 -11988.403,E2 -11988.403} C_VEL
LIN {X 0,Y 389.255,Z 284.984,A -85,B 0,C 180,E1 -11988.759,E2 -11988.759} C_VEL
LIN {X 0,Y 389.962,Z 218.396,A -85,B 0,C 180,E1 -11989.996,E2 -11989.996} C_VEL
LIN {X 0,Y 385.435,Z 189.959,A -85,B 0,C 180,E1 -11990.79,E2 -11990.79} C_VEL
LIN {X 0,Y 385.102,Z 187.928,A -85,B 0,C 180,E1 -11990.868,E2 -11990.868} C_VEL
LIN {X 0,Y 386.613,Z 170.128,A -85,B 0,C 180,E1 -11994.643,E2 -11994.643} C_VEL
LIN {X 0,Y 386.158,Z 165.855,A -85,B 0,C 180,E1 -11995.609,E2 -11995.609} C_VEL
LIN {X 0,Y 383.457,Z 152.625,A -85,B 0,C 180,E1 -11998.756,E2 -11998.756} C_VEL
LIN {X 0,Y 383.019,Z 150.776,A -85,B 0,C 180,E1 -11999.243,E2 -11999.243} C_VEL
LIN {X 0,Y 382.982,Z 150.776,A -85,B 0,C 180,E1 -12002.421,E2 -12002.421} C_VEL
LIN {X 0,Y 383.019,Z 150.773,A -85,B 0,C 180,E1 -12005.955,E2 -12005.955} C_VEL
LIN {X 0,Y 382.981,Z 150.78,A -85,B 0,C 180,E1 -12009.58,E2 -12009.58} C_VEL
LIN {X 0,Y 383.001,Z 150.775,A -85,B 0,C 180,E1 -12012.778,E2 -12012.778} C_VEL
LIN {X 0,Y 382.984,Z 150.776,A -85,B 0,C 180,E1 -12015.787,E2 -12015.787} C_VEL
LIN {X 0,Y 382.955,Z 150.782,A -85,B 0,C 180,E1 -12018.8,E2 -12018.8} C_VEL
LIN {X 0,Y 382.987,Z 150.775,A -85,B 0,C 180,E1 -12022.097,E2 -12022.097} C_VEL
LIN {X 0,Y 383.004,Z 150.775,A -85,B 0,C 180,E1 -12025.331,E2 -12025.331} C_VEL
LIN {X 0,Y 382.973,Z 150.78,A -85,B 0,C 180,E1 -12029.08,E2 -12029.08} C_VEL
LIN {X 0,Y 382.973,Z 150.783,A -85,B 0,C 180,E1 -12032.692,E2 -12032.692} C_VEL
LIN {X 0,Y 383.001,Z 150.775,A -85,B 0,C 180,E1 -12036.191,E2 -12036.191} C_VEL
LIN {X 0,Y 383.032,Z 150.769,A -85,B 0,C 180,E1 -12039.597,E2 -12039.597} C_VEL
LIN {X 0,Y 383.06,Z 150.768,A -85,B 0,C 180,E1 -12042.929,E2 -12042.929} C_VEL
LIN {X 0,Y 383.117,Z 150.764,A -85,B 0,C 180,E1 -12046.464,E2 -12046.464} C_VEL
LIN {X 0,Y 383.126,Z 150.761,A -85,B 0,C 180,E1 -12050.497,E2 -12050.497} C_VEL
LIN {X 0,Y 383.222,Z 150.748,A -85,B 0,C 180,E1 -12053.683,E2 -12053.683} C_VEL
LIN {X 0,Y 383.358,Z 150.734,A -85,B 0,C 180,E1 -12057.899,E2 -12057.899} C_VEL
LIN {X 0,Y 383.362,Z 150.733,A -85,B 0,C 180,E1 -12062.101,E2 -12062.101} C_VEL
LIN {X 0,Y 383.22,Z 150.747,A -85,B 0,C 180,E1 -12066.419,E2 -12066.419} C_VEL
LIN {X 0,Y 383.133,Z 150.761,A -85,B 0,C 180,E1 -12069.503,E2 -12069.503} C_VEL
LIN {X 0,Y 383.117,Z 150.765,A -85,B 0,C 180,E1 -12073.536,E2 -12073.536} C_VEL
LIN {X 0,Y 383.044,Z 150.774,A -85,B 0,C 180,E1 -12077.435,E2 -12077.435} C_VEL
LIN {X 0,Y 383.023,Z 150.771,A -85,B 0,C 180,E1 -12080.648,E2 -12080.648} C_VEL
LIN {X 0,Y 383.002,Z 150.775,A -85,B 0,C 180,E1 -12083.81,E2 -12083.81} C_VEL
LIN {X 0,Y 382.977,Z 150.782,A -85,B 0,C 180,E1 -12087.308,E2 -12087.308} C_VEL
LIN {X 0,Y 382.974,Z 150.781,A -85,B 0,C 180,E1 -12090.92,E2 -12090.92} C_VEL
LIN {X 0,Y 383.005,Z 150.776,A -85,B 0,C 180,E1 -12094.67,E2 -12094.67} C_VEL
LIN {X 0,Y 382.988,Z 150.775,A -85,B 0,C 180,E1 -12097.903,E2 -12097.903} C_VEL
LIN {X 0,Y 382.956,Z 150.78,A -85,B 0,C 180,E1 -12101.351,E2 -12101.351} C_VEL
LIN {X 0,Y 382.989,Z 150.777,A -85,B 0,C 180,E1 -12104.304,E2 -12104.304} C_VEL
LIN {X 0,Y 383.006,Z 150.774,A -85,B 0,C 180,E1 -12107.241,E2 -12107.241} C_VEL
LIN {X 0,Y 382.989,Z 150.78,A -85,B 0,C 180,E1 -12110.419,E2 -12110.419} C_VEL
LIN {X 0,Y 383.021,Z 150.773,A -85,B 0,C 180,E1 -12114.045,E2 -12114.045} C_VEL
LIN {X 0,Y 382.985,Z 150.775,A -85,B 0,C 180,E1 -12117.579,E2 -12117.579} C_VEL
LIN {X 0,Y 382.978,Z 150.783,A -85,B 0,C 180,E1 -12120.3,E2 -12120.3} C_VEL
LIN {X 0,Y 383.003,Z 150.778,A -85,B 0,C 180,E1 -12124.045,E2 -12124.045} C_VEL
LIN {X 0,Y 383.048,Z 150.779,A -85,B 0,C 180,E1 -12126.252,E2 -12126.252} C_VEL
LIN {X 0,Y 385.418,Z 162.469,A -85,B 0,C 180,E1 -12129.231,E2 -12129.231} C_VEL
LIN {X 0,Y 387.63,Z 170.758,A -85,B 0,C 180,E1 -12129.518,E2 -12129.518} C_VEL
LIN {X 0,Y 390.578,Z 185.389,A -85,B 0,C 180,E1 -12129.963,E2 -12129.963} C_VEL
LIN {X 0,Y 389.424,Z 265.975,A -85,B 0,C 180,E1 -12131.454,E2 -12131.454} C_VEL
LIN {X 0,Y 389.046,Z 279.218,A -85,B 0,C 180,E1 -12131.844,E2 -12131.844} C_VEL
LIN {X 0,Y 388.466,Z 291.808,A -85,B 0,C 180,E1 -12132.429,E2 -12132.429} C_VEL
LIN {X 0,Y 387.749,Z 303.032,A -85,B 0,C 180,E1 -12133.143,E2 -12133.143} C_VEL
LIN {X 0,Y 386.915,Z 314.126,A -85,B 0,C 180,E1 -12134.055,E2 -12134.055} C_VEL
LIN {X 0,Y 386.155,Z 325.422,A -85,B 0,C 180,E1 -12135.239,E2 -12135.239} C_VEL
LIN {X 0,Y 385.096,Z 335.393,A -85,B 0,C 180,E1 -12136.545,E2 -12136.545} C_VEL
LIN {X 0,Y 384.334,Z 343.548,A -85,B 0,C 180,E1 -12137.861,E2 -12137.861} C_VEL
LIN {X 0,Y 383.501,Z 351.539,A -85,B 0,C 180,E1 -12139.441,E2 -12139.441} C_VEL
LIN {X 0,Y 382.83,Z 357.951,A -85,B 0,C 180,E1 -12141.023,E2 -12141.023} C_VEL
LIN {X 0,Y 382.415,Z 363.034,A -85,B 0,C 180,E1 -12142.609,E2 -12142.609} C_VEL
LIN {X 0,Y 382.117,Z 366.98,A -85,B 0,C 180,E1 -12144.195,E2 -12144.195} C_VEL
LIN {X 0,Y 381.829,Z 369.898,A -85,B 0,C 180,E1 -12145.778,E2 -12145.778} C_VEL
LIN {X 0,Y 381.787,Z 371.293,A -85,B 0,C 180,E1 -12146.835,E2 -12146.835} C_VEL
LIN {X 0,Y 381.743,Z 372.285,A -85,B 0,C 180,E1 -12147.89,E2 -12147.89} C_VEL
LIN {X 0,Y 381.662,Z 373.131,A -85,B 0,C 180,E1 -12150.001,E2 -12150.001} C_VEL
LIN {X 0,Y 381.683,Z 372.942,A -85,B 0,C 180,E1 -12151.056,E2 -12151.056} C_VEL
LIN {X 0,Y 381.743,Z 372.358,A -85,B 0,C 180,E1 -12152.111,E2 -12152.111} C_VEL
LIN {X 0,Y 381.782,Z 371.394,A -85,B 0,C 180,E1 -12153.166,E2 -12153.166} C_VEL
LIN {X 0,Y 381.819,Z 370.044,A -85,B 0,C 180,E1 -12154.223,E2 -12154.223} C_VEL
LIN {X 0,Y 382.108,Z 367.181,A -85,B 0,C 180,E1 -12155.806,E2 -12155.806} C_VEL
LIN {X 0,Y 382.358,Z 363.018,A -85,B 0,C 180,E1 -12157.491,E2 -12157.491} C_VEL
LIN {X 0,Y 382.784,Z 358.3,A -85,B 0,C 180,E1 -12158.979,E2 -12158.979} C_VEL
LIN {X 0,Y 383.471,Z 351.994,A -85,B 0,C 180,E1 -12160.561,E2 -12160.561} C_VEL
LIN {X 0,Y 383.868,Z 347.656,A -85,B 0,C 180,E1 -12161.472,E2 -12161.472} C_VEL
LIN {X 0,Y 383.632,Z 344.097,A -85,B 0,C 180,E1 -12162.17,E2 -12162.17} C_VEL
LIN {X 0,Y 381.515,Z 338.032,A -85,B 0,C 180,E1 -12163.3,E2 -12163.3} C_VEL
LIN {X 0,Y 379.395,Z 331.452,A -85,B 0,C 180,E1 -12164.372,E2 -12164.372} C_VEL
LIN {X 0,Y 379.153,Z 327.021,A -85,B 0,C 180,E1 -12164.971,E2 -12164.971} C_VEL
LIN {X 0,Y 379.957,Z 316.815,A -85,B 0,C 180,E1 -12166.109,E2 -12166.109} C_VEL
LIN {X 0,Y 380.815,Z 306.347,A -85,B 0,C 180,E1 -12167.036,E2 -12167.036} C_VEL
LIN {X 0,Y 381.592,Z 294.862,A -85,B 0,C 180,E1 -12167.83,E2 -12167.83} C_VEL
LIN {X 0,Y 382.296,Z 281.868,A -85,B 0,C 180,E1 -12168.489,E2 -12168.489} C_VEL
LIN {X 0,Y 382.776,Z 269.122,A -85,B 0,C 180,E1 -12168.916,E2 -12168.916} C_VEL
LIN {X 0,Y 383.916,Z 186.305,A -85,B 0,C 180,E1 -12170.491,E2 -12170.491} C_VEL
LIN {X 0,Y 379.829,Z 167.161,A -85,B 0,C 180,E1 -12171.104,E2 -12171.104} C_VEL
LIN {X 0,Y 378.185,Z 162.444,A -85,B 0,C 180,E1 -12171.312,E2 -12171.312} C_VEL
LIN {X 0,Y 375.995,Z 151.651,A -85,B 0,C 180,E1 -12174.197,E2 -12174.197} C_VEL
LIN {X 0,Y 375.938,Z 151.66,A -85,B 0,C 180,E1 -12177.864,E2 -12177.864} C_VEL
LIN {X 0,Y 375.96,Z 151.655,A -85,B 0,C 180,E1 -12181.562,E2 -12181.562} C_VEL
LIN {X 0,Y 375.959,Z 151.655,A -85,B 0,C 180,E1 -12185.415,E2 -12185.415} C_VEL
LIN {X 0,Y 375.936,Z 151.654,A -85,B 0,C 180,E1 -12188.263,E2 -12188.263} C_VEL
LIN {X 0,Y 375.92,Z 151.66,A -85,B 0,C 180,E1 -12191.598,E2 -12191.598} C_VEL
LIN {X 0,Y 375.927,Z 151.655,A -85,B 0,C 180,E1 -12194.731,E2 -12194.731} C_VEL
LIN {X 0,Y 375.926,Z 151.657,A -85,B 0,C 180,E1 -12197.699,E2 -12197.699} C_VEL
LIN {X 0,Y 375.935,Z 151.654,A -85,B 0,C 180,E1 -12200.534,E2 -12200.534} C_VEL
LIN {X 0,Y 375.958,Z 151.653,A -85,B 0,C 180,E1 -12203.497,E2 -12203.497} C_VEL
LIN {X 0,Y 375.957,Z 151.651,A -85,B 0,C 180,E1 -12205.888,E2 -12205.888} C_VEL
LIN {X 0,Y 375.96,Z 151.651,A -85,B 0,C 180,E1 -12209.687,E2 -12209.687} C_VEL
LIN {X 0,Y 375.928,Z 151.655,A -85,B 0,C 180,E1 -12212.136,E2 -12212.136} C_VEL
LIN {X 0,Y 375.972,Z 151.649,A -85,B 0,C 180,E1 -12215.717,E2 -12215.717} C_VEL
LIN {X 0,Y 375.997,Z 151.647,A -85,B 0,C 180,E1 -12219.198,E2 -12219.198} C_VEL
LIN {X 0,Y 376.007,Z 151.651,A -85,B 0,C 180,E1 -12222.599,E2 -12222.599} C_VEL
LIN {X 0,Y 376.088,Z 151.639,A -85,B 0,C 180,E1 -12226.342,E2 -12226.342} C_VEL
LIN {X 0,Y 376.11,Z 151.638,A -85,B 0,C 180,E1 -12230.318,E2 -12230.318} C_VEL
LIN {X 0,Y 376.19,Z 151.622,A -85,B 0,C 180,E1 -12233.564,E2 -12233.564} C_VEL
LIN {X 0,Y 376.334,Z 151.607,A -85,B 0,C 180,E1 -12237.859,E2 -12237.859} C_VEL
LIN {X 0,Y 376.329,Z 151.609,A -85,B 0,C 180,E1 -12242.14,E2 -12242.14} C_VEL
LIN {X 0,Y 376.189,Z 151.623,A -85,B 0,C 180,E1 -12246.436,E2 -12246.436} C_VEL
LIN {X 0,Y 376.103,Z 151.638,A -85,B 0,C 180,E1 -12249.682,E2 -12249.682} C_VEL
LIN {X 0,Y 376.038,Z 151.646,A -85,B 0,C 180,E1 -12253.626,E2 -12253.626} C_VEL
LIN {X 0,Y 375.98,Z 151.654,A -85,B 0,C 180,E1 -12257.577,E2 -12257.577} C_VEL
LIN {X 0,Y 375.977,Z 151.649,A -85,B 0,C 180,E1 -12260.832,E2 -12260.832} C_VEL
LIN {X 0,Y 375.932,Z 151.654,A -85,B 0,C 180,E1 -12264.286,E2 -12264.286} C_VEL
LIN {X 0,Y 375.908,Z 151.657,A -85,B 0,C 180,E1 -12266.661,E2 -12266.661} C_VEL
LIN {X 0,Y 375.91,Z 151.661,A -85,B 0,C 180,E1 -12269.084,E2 -12269.084} C_VEL
LIN {X 0,Y 375.952,Z 151.654,A -85,B 0,C 180,E1 -12271.563,E2 -12271.563} C_VEL
LIN {X 0,Y 375.948,Z 151.655,A -85,B 0,C 180,E1 -12275.417,E2 -12275.417} C_VEL
LIN {X 0,Y 375.936,Z 151.654,A -85,B 0,C 180,E1 -12278.263,E2 -12278.263} C_VEL
LIN {X 0,Y 375.916,Z 151.656,A -85,B 0,C 180,E1 -12281.598,E2 -12281.598} C_VEL
LIN {X 0,Y 375.921,Z 151.661,A -85,B 0,C 180,E1 -12284.73,E2 -12284.73} C_VEL
LIN {X 0,Y 375.907,Z 151.657,A -85,B 0,C 180,E1 -12287.696,E2 -12287.696} C_VEL
LIN {X 0,Y 375.935,Z 151.659,A -85,B 0,C 180,E1 -12290.534,E2 -12290.534} C_VEL
LIN {X 0,Y 375.963,Z 151.65,A -85,B 0,C 180,E1 -12293.496,E2 -12293.496} C_VEL
LIN {X 0,Y 375.96,Z 151.651,A -85,B 0,C 180,E1 -12295.888,E2 -12295.888} C_VEL
LIN {X 0,Y 375.965,Z 151.655,A -85,B 0,C 180,E1 -12299.687,E2 -12299.687} C_VEL
LIN {X 0,Y 375.973,Z 151.738,A -85,B 0,C 180,E1 -12300.46,E2 -12300.46} C_VEL
LIN {X 0,Y 378.289,Z 162.432,A -85,B 0,C 180,E1 -12303.096,E2 -12303.096} C_VEL
LIN {X 0,Y 379.697,Z 170.873,A -85,B 0,C 180,E1 -12305.09,E2 -12305.09} C_VEL
LIN {X 0,Y 378.264,Z 187.662,A -85,B 0,C 180,E1 -12308.723,E2 -12308.723} C_VEL
LIN {X 0,Y 383.112,Z 217.726,A -85,B 0,C 180,E1 -12309.611,E2 -12309.611} C_VEL
LIN {X 0,Y 383.463,Z 223.039,A -85,B 0,C 180,E1 -12309.734,E2 -12309.734} C_VEL
LIN {X 0,Y 382.335,Z 296.408,A -85,B 0,C 180,E1 -12311.131,E2 -12311.131} C_VEL
LIN {X 0,Y 381.714,Z 309.627,A -85,B 0,C 180,E1 -12311.586,E2 -12311.586} C_VEL
LIN {X 0,Y 380.885,Z 321.764,A -85,B 0,C 180,E1 -12312.205,E2 -12312.205} C_VEL
LIN {X 0,Y 379.924,Z 334.017,A -85,B 0,C 180,E1 -12313.061,E2 -12313.061} C_VEL
LIN {X 0,Y 378.832,Z 345.611,A -85,B 0,C 180,E1 -12314.119,E2 -12314.119} C_VEL
LIN {X 0,Y 377.881,Z 356.457,A -85,B 0,C 180,E1 -12315.372,E2 -12315.372} C_VEL
LIN {X 0,Y 376.962,Z 366.282,A -85,B 0,C 180,E1 -12316.798,E2 -12316.798} C_VEL
LIN {X 0,Y 375.959,Z 375.226,A -85,B 0,C 180,E1 -12318.407,E2 -12318.407} C_VEL
LIN {X 0,Y 375.328,Z 382.432,A -85,B 0,C 180,E1 -12320.025,E2 -12320.025} C_VEL
LIN {X 0,Y 374.993,Z 387.3,A -85,B 0,C 180,E1 -12321.377,E2 -12321.377} C_VEL
LIN {X 0,Y 374.672,Z 392.032,A -85,B 0,C 180,E1 -12322.996,E2 -12322.996} C_VEL
LIN {X 0,Y 374.534,Z 395.65,A -85,B 0,C 180,E1 -12324.616,E2 -12324.616} C_VEL
LIN {X 0,Y 374.547,Z 397.519,A -85,B 0,C 180,E1 -12325.695,E2 -12325.695} C_VEL
LIN {X 0,Y 374.499,Z 399.918,A -85,B 0,C 180,E1 -12327.848,E2 -12327.848} C_VEL
LIN {X 0,Y 374.569,Z 400.53,A -85,B 0,C 180,E1 -12328.924,E2 -12328.924} C_VEL
LIN {X 0,Y 374.592,Z 400.746,A -85,B 0,C 180,E1 -12329.999,E2 -12329.999} C_VEL
LIN {X 0,Y 374.568,Z 400.526,A -85,B 0,C 180,E1 -12331.075,E2 -12331.075} C_VEL
LIN {X 0,Y 374.465,Z 398.91,A -85,B 0,C 180,E1 -12333.227,E2 -12333.227} C_VEL
LIN {X 0,Y 374.55,Z 397.508,A -85,B 0,C 180,E1 -12334.304,E2 -12334.304} C_VEL
LIN {X 0,Y 374.58,Z 394.254,A -85,B 0,C 180,E1 -12336.062,E2 -12336.062} C_VEL
LIN {X 0,Y 374.771,Z 390.568,A -85,B 0,C 180,E1 -12337.542,E2 -12337.542} C_VEL
LIN {X 0,Y 375.172,Z 384.437,A -85,B 0,C 180,E1 -12339.433,E2 -12339.433} C_VEL
LIN {X 0,Y 375.721,Z 377.742,A -85,B 0,C 180,E1 -12341.053,E2 -12341.053} C_VEL
LIN {X 0,Y 376.597,Z 369.445,A -85,B 0,C 180,E1 -12342.666,E2 -12342.666} C_VEL
LIN {X 0,Y 377.572,Z 359.769,A -85,B 0,C 180,E1 -12344.168,E2 -12344.168} C_VEL
LIN {X 0,Y 378.485,Z 349.253,A -85,B 0,C 180,E1 -12345.481,E2 -12345.481} C_VEL
LIN {X 0,Y 379.454,Z 338.609,A -85,B 0,C 180,E1 -12346.544,E2 -12346.544} C_VEL
LIN {X 0,Y 380.511,Z 326.72,A -85,B 0,C 180,E1 -12347.465,E2 -12347.465} C_VEL
LIN {X 0,Y 381.353,Z 314.348,A -85,B 0,C 180,E1 -12348.188,E2 -12348.188} C_VEL
LIN {X 0,Y 382.096,Z 301.639,A -85,B 0,C 180,E1 -12348.706,E2 -12348.706} C_VEL
LIN {X 0,Y 382.502,Z 288.287,A -85,B 0,C 180,E1 -12349.033,E2 -12349.033} C_VEL
LIN {X 0,Y 383.293,Z 219.346,A -85,B 0,C 180,E1 -12350.335,E2 -12350.335} C_VEL
LIN {X 0,Y 378.942,Z 191.855,A -85,B 0,C 180,E1 -12351.12,E2 -12351.12} C_VEL
LIN {X 0,Y 378.236,Z 187.604,A -85,B 0,C 180,E1 -12351.278,E2 -12351.278} C_VEL
LIN {X 0,Y 379.581,Z 172.786,A -85,B 0,C 180,E1 -12354.476,E2 -12354.476} C_VEL
LIN {X 0,Y 379.618,Z 169.53,A -85,B 0,C 180,E1 -12355.201,E2 -12355.201} C_VEL
LIN {X 0,Y 377.104,Z 156.662,A -85,B 0,C 180,E1 -12358.294,E2 -12358.294} C_VEL
LIN {X 0,Y 375.964,Z 151.656,A -85,B 0,C 180,E1 -12359.578,E2 -12359.578} C_VEL
LIN {X 0,Y 375.945,Z 151.653,A -85,B 0,C 180,E1 -12362.828,E2 -12362.828} C_VEL
LIN {X 0,Y 375.952,Z 151.657,A -85,B 0,C 180,E1 -12365.415,E2 -12365.415} C_VEL
LIN {X 0,Y 375.931,Z 151.654,A -85,B 0,C 180,E1 -12368.262,E2 -12368.262} C_VEL
LIN {X 0,Y 375.913,Z 151.66,A -85,B 0,C 180,E1 -12371.597,E2 -12371.597} C_VEL
LIN {X 0,Y 375.919,Z 151.657,A -85,B 0,C 180,E1 -12374.73,E2 -12374.73} C_VEL
LIN {X 0,Y 375.919,Z 151.657,A -85,B 0,C 180,E1 -12377.698,E2 -12377.698} C_VEL
LIN {X 0,Y 375.929,Z 151.656,A -85,B 0,C 180,E1 -12380.533,E2 -12380.533} C_VEL
LIN {X 0,Y 375.951,Z 151.653,A -85,B 0,C 180,E1 -12383.496,E2 -12383.496} C_VEL
LIN {X 0,Y 375.95,Z 151.651,A -85,B 0,C 180,E1 -12385.887,E2 -12385.887} C_VEL
LIN {X 0,Y 375.953,Z 151.651,A -85,B 0,C 180,E1 -12389.686,E2 -12389.686} C_VEL
LIN {X 0,Y 375.917,Z 151.657,A -85,B 0,C 180,E1 -12392.135,E2 -12392.135} C_VEL
LIN {X 0,Y 375.928,Z 151.659,A -85,B 0,C 180,E1 -12394.533,E2 -12394.533} C_VEL
LIN {X 0,Y 375.965,Z 151.653,A -85,B 0,C 180,E1 -12396.886,E2 -12396.886} C_VEL
LIN {X 0,Y 375.965,Z 151.654,A -85,B 0,C 180,E1 -12400.338,E2 -12400.338} C_VEL
LIN {X 0,Y 375.964,Z 151.65,A -85,B 0,C 180,E1 -12403.716,E2 -12403.716} C_VEL
LIN {X 0,Y 376.093,Z 151.634,A -85,B 0,C 180,E1 -12407.042,E2 -12407.042} C_VEL
LIN {X 0,Y 376.097,Z 151.639,A -85,B 0,C 180,E1 -12410.318,E2 -12410.318} C_VEL
LIN {X 0,Y 376.182,Z 151.624,A -85,B 0,C 180,E1 -12413.564,E2 -12413.564} C_VEL
LIN {X 0,Y 376.322,Z 151.61,A -85,B 0,C 180,E1 -12417.859,E2 -12417.859} C_VEL
LIN {X 0,Y 376.327,Z 151.608,A -85,B 0,C 180,E1 -12422.141,E2 -12422.141} C_VEL
LIN {X 0,Y 376.188,Z 151.623,A -85,B 0,C 180,E1 -12426.436,E2 -12426.436} C_VEL
LIN {X 0,Y 376.103,Z 151.639,A -85,B 0,C 180,E1 -12429.682,E2 -12429.682} C_VEL
LIN {X 0,Y 376.081,Z 151.641,A -85,B 0,C 180,E1 -12433.658,E2 -12433.658} C_VEL
LIN {X 0,Y 375.998,Z 151.651,A -85,B 0,C 180,E1 -12437.59,E2 -12437.59} C_VEL
LIN {X 0,Y 375.971,Z 151.65,A -85,B 0,C 180,E1 -12440.833,E2 -12440.833} C_VEL
LIN {X 0,Y 375.928,Z 151.654,A -85,B 0,C 180,E1 -12444.286,E2 -12444.286} C_VEL
LIN {X 0,Y 375.914,Z 151.657,A -85,B 0,C 180,E1 -12446.66,E2 -12446.66} C_VEL
LIN {X 0,Y 375.909,Z 151.662,A -85,B 0,C 180,E1 -12449.084,E2 -12449.084} C_VEL
LIN {X 0,Y 375.949,Z 151.653,A -85,B 0,C 180,E1 -12451.563,E2 -12451.563} C_VEL
LIN {X 0,Y 375.943,Z 151.654,A -85,B 0,C 180,E1 -12455.417,E2 -12455.417} C_VEL
LIN {X 0,Y 375.931,Z 151.655,A -85,B 0,C 180,E1 -12458.264,E2 -12458.264} C_VEL
LIN {X 0,Y 375.912,Z 151.656,A -85,B 0,C 180,E1 -12461.599,E2 -12461.599} C_VEL
LIN {X 0,Y 375.921,Z 151.662,A -85,B 0,C 180,E1 -12464.732,E2 -12464.732} C_VEL
LIN {X 0,Y 375.919,Z 151.659,A -85,B 0,C 180,E1 -12468.402,E2 -12468.402} C_VEL
LIN {X 0,Y 375.934,Z 151.654,A -85,B 0,C 180,E1 -12471.738,E2 -12471.738} C_VEL
LIN {X 0,Y 375.977,Z 151.648,A -85,B 0,C 180,E1 -12475.334,E2 -12475.334} C_VEL
LIN {X 0,Y 375.955,Z 151.656,A -85,B 0,C 180,E1 -12478.439,E2 -12478.439} C_VEL
LIN {X 0,Y 375.932,Z 151.659,A -85,B 0,C 180,E1 -12482.137,E2 -12482.137} C_VEL
LIN {X 0,Y 375.992,Z 151.653,A -85,B 0,C 180,E1 -12485.939,E2 -12485.939} C_VEL
LIN {X 0,Y 378.261,Z 162.562,A -85,B 0,C 180,E1 -12488.815,E2 -12488.815} C_VEL
LIN {X 0,Y 380.648,Z 170.297,A -85,B 0,C 180,E1 -12489.11,E2 -12489.11} C_VEL
LIN {X 0,Y 383.882,Z 186.129,A -85,B 0,C 180,E1 -12489.607,E2 -12489.607} C_VEL
LIN {X 0,Y 382.7,Z 266.255,A -85,B 0,C 180,E1 -12491.116,E2 -12491.116} C_VEL
LIN {X 0,Y 382.323,Z 279.49,A -85,B 0,C 180,E1 -12491.514,E2 -12491.514} C_VEL
LIN {X 0,Y 381.714,Z 292.075,A -85,B 0,C 180,E1 -12492.108,E2 -12492.108} C_VEL
LIN {X 0,Y 380.959,Z 303.297,A -85,B 0,C 180,E1 -12492.833,E2 -12492.833} C_VEL
LIN {X 0,Y 380.096,Z 314.39,A -85,B 0,C 180,E1 -12493.761,E2 -12493.761} C_VEL
LIN {X 0,Y 379.307,Z 325.684,A -85,B 0,C 180,E1 -12494.966,E2 -12494.966} C_VEL
LIN {X 0,Y 378.208,Z 335.655,A -85,B 0,C 180,E1 -12496.296,E2 -12496.296} C_VEL
LIN {X 0,Y 377.392,Z 343.81,A -85,B 0,C 180,E1 -12497.635,E2 -12497.635} C_VEL
LIN {X 0,Y 376.51,Z 351.8,A -85,B 0,C 180,E1 -12499.243,E2 -12499.243} C_VEL
LIN {X 0,Y 375.816,Z 358.212,A -85,B 0,C 180,E1 -12500.854,E2 -12500.854} C_VEL
LIN {X 0,Y 375.372,Z 363.294,A -85,B 0,C 180,E1 -12502.47,E2 -12502.47} C_VEL
LIN {X 0,Y 375.057,Z 367.24,A -85,B 0,C 180,E1 -12504.085,E2 -12504.085} C_VEL
LIN {X 0,Y 374.758,Z 370.157,A -85,B 0,C 180,E1 -12505.699,E2 -12505.699} C_VEL
LIN {X 0,Y 374.695,Z 371.553,A -85,B 0,C 180,E1 -12506.775,E2 -12506.775} C_VEL
LIN {X 0,Y 374.649,Z 372.545,A -85,B 0,C 180,E1 -12507.85,E2 -12507.85} C_VEL
LIN {X 0,Y 374.594,Z 373.389,A -85,B 0,C 180,E1 -12510.001,E2 -12510.001} C_VEL
LIN {X 0,Y 374.6,Z 373.201,A -85,B 0,C 180,E1 -12511.076,E2 -12511.076} C_VEL
LIN {X 0,Y 374.649,Z 372.617,A -85,B 0,C 180,E1 -12512.151,E2 -12512.151} C_VEL
LIN {X 0,Y 374.749,Z 370.302,A -85,B 0,C 180,E1 -12514.303,E2 -12514.303} C_VEL
LIN {X 0,Y 375.047,Z 367.439,A -85,B 0,C 180,E1 -12515.916,E2 -12515.916} C_VEL
LIN {X 0,Y 375.294,Z 363.563,A -85,B 0,C 180,E1 -12517.533,E2 -12517.533} C_VEL
LIN {X 0,Y 375.778,Z 358.557,A -85,B 0,C 180,E1 -12519.148,E2 -12519.148} C_VEL
LIN {X 0,Y 376.479,Z 352.252,A -85,B 0,C 180,E1 -12520.759,E2 -12520.759} C_VEL
LIN {X 0,Y 377.297,Z 344.359,A -85,B 0,C 180,E1 -12522.37,E2 -12522.37} C_VEL
LIN {X 0,Y 378.189,Z 336.308,A -85,B 0,C 180,E1 -12523.706,E2 -12523.706} C_VEL
LIN {X 0,Y 379.153,Z 327.021,A -85,B 0,C 180,E1 -12524.971,E2 -12524.971} C_VEL
LIN {X 0,Y 378.901,Z 322.477,A -85,B 0,C 180,E1 -12525.543,E2 -12525.543} C_VEL
LIN {X 0,Y 376.755,Z 314.905,A -85,B 0,C 180,E1 -12526.46,E2 -12526.46} C_VEL
LIN {X 0,Y 374.666,Z 306.934,A -85,B 0,C 180,E1 -12527.295,E2 -12527.295} C_VEL
LIN {X 0,Y 374.368,Z 301.75,A -85,B 0,C 180,E1 -12527.724,E2 -12527.724} C_VEL
LIN {X 0,Y 375.184,Z 289.185,A -85,B 0,C 180,E1 -12528.499,E2 -12528.499} C_VEL
LIN {X 0,Y 375.81,Z 276.023,A -85,B 0,C 180,E1 -12529.068,E2 -12529.068} C_VEL
LIN {X 0,Y 376.218,Z 263.221,A -85,B 0,C 180,E1 -12529.401,E2 -12529.401} C_VEL
LIN {X 0,Y 377.291,Z 187.337,A -85,B 0,C 180,E1 -12530.851,E2 -12530.851} C_VEL
LIN {X 0,Y 373.46,Z 169.43,A -85,B 0,C 180,E1 -12531.441,E2 -12531.441} C_VEL
LIN {X 0,Y 371.041,Z 162.626,A -85,B 0,C 180,E1 -12531.764,E2 -12531.764} C_VEL
LIN {X 0,Y 368.936,Z 152.528,A -85,B 0,C 180,E1 -12534.545,E2 -12534.545} C_VEL
LIN {X 0,Y 368.878,Z 152.535,A -85,B 0,C 180,E1 -12537.21,E2 -12537.21} C_VEL
LIN {X 0,Y 368.931,Z 152.526,A -85,B 0,C 180,E1 -12540.953,E2 -12540.953} C_VEL
LIN {X 0,Y 368.93,Z 152.527,A -85,B 0,C 180,E1 -12545.001,E2 -12545.001} C_VEL
LIN {X 0,Y 368.878,Z 152.533,A -85,B 0,C 180,E1 -12548.634,E2 -12548.634} C_VEL
LIN {X 0,Y 368.872,Z 152.534,A -85,B 0,C 180,E1 -12552.007,E2 -12552.007} C_VEL
LIN {X 0,Y 368.88,Z 152.537,A -85,B 0,C 180,E1 -12555.175,E2 -12555.175} C_VEL
LIN {X 0,Y 368.87,Z 152.533,A -85,B 0,C 180,E1 -12558.176,E2 -12558.176} C_VEL
LIN {X 0,Y 368.877,Z 152.537,A -85,B 0,C 180,E1 -12561.366,E2 -12561.366} C_VEL
LIN {X 0,Y 368.93,Z 152.532,A -85,B 0,C 180,E1 -12565.146,E2 -12565.146} C_VEL
LIN {X 0,Y 368.912,Z 152.534,A -85,B 0,C 180,E1 -12569.045,E2 -12569.045} C_VEL
LIN {X 0,Y 368.911,Z 152.529,A -85,B 0,C 180,E1 -12571.558,E2 -12571.558} C_VEL
LIN {X 0,Y 368.925,Z 152.529,A -85,B 0,C 180,E1 -12575.222,E2 -12575.222} C_VEL
LIN {X 0,Y 368.919,Z 152.531,A -85,B 0,C 180,E1 -12578.98,E2 -12578.98} C_VEL
LIN {X 0,Y 368.952,Z 152.526,A -85,B 0,C 180,E1 -12582.255,E2 -12582.255} C_VEL
LIN {X 0,Y 369.036,Z 152.517,A -85,B 0,C 180,E1 -12586.228,E2 -12586.228} C_VEL
LIN {X 0,Y 369.06,Z 152.514,A -85,B 0,C 180,E1 -12590.131,E2 -12590.131} C_VEL
LIN {X 0,Y 369.151,Z 152.499,A -85,B 0,C 180,E1 -12593.441,E2 -12593.441} C_VEL
LIN {X 0,Y 369.298,Z 152.483,A -85,B 0,C 180,E1 -12597.819,E2 -12597.819} C_VEL
LIN {X 0,Y 369.292,Z 152.485,A -85,B 0,C 180,E1 -12602.181,E2 -12602.181} C_VEL
LIN {X 0,Y 369.152,Z 152.499,A -85,B 0,C 180,E1 -12606.559,E2 -12606.559} C_VEL
LIN {X 0,Y 369.054,Z 152.516,A -85,B 0,C 180,E1 -12609.869,E2 -12609.869} C_VEL
LIN {X 0,Y 368.999,Z 152.523,A -85,B 0,C 180,E1 -12613.749,E2 -12613.749} C_VEL
LIN {X 0,Y 368.934,Z 152.53,A -85,B 0,C 180,E1 -12617.746,E2 -12617.746} C_VEL
LIN {X 0,Y 368.907,Z 152.533,A -85,B 0,C 180,E1 -12621.221,E2 -12621.221} C_VEL
LIN {X 0,Y 368.905,Z 152.531,A -85,B 0,C 180,E1 -12623.873,E2 -12623.873} C_VEL
LIN {X 0,Y 368.855,Z 152.541,A -85,B 0,C 180,E1 -12627.212,E2 -12627.212} C_VEL
LIN {X 0,Y 368.89,Z 152.533,A -85,B 0,C 180,E1 -12629.693,E2 -12629.693} C_VEL
LIN {X 0,Y 368.894,Z 152.536,A -85,B 0,C 180,E1 -12633.043,E2 -12633.043} C_VEL
LIN {X 0,Y 368.911,Z 152.529,A -85,B 0,C 180,E1 -12636.198,E2 -12636.198} C_VEL
LIN {X 0,Y 368.874,Z 152.539,A -85,B 0,C 180,E1 -12638.957,E2 -12638.957} C_VEL
LIN {X 0,Y 368.87,Z 152.534,A -85,B 0,C 180,E1 -12642.007,E2 -12642.007} C_VEL
LIN {X 0,Y 368.873,Z 152.536,A -85,B 0,C 180,E1 -12645.175,E2 -12645.175} C_VEL
LIN {X 0,Y 368.86,Z 152.536,A -85,B 0,C 180,E1 -12648.174,E2 -12648.174} C_VEL
LIN {X 0,Y 368.877,Z 152.533,A -85,B 0,C 180,E1 -12651.366,E2 -12651.366} C_VEL
LIN {X 0,Y 368.936,Z 152.526,A -85,B 0,C 180,E1 -12655.146,E2 -12655.146} C_VEL
LIN {X 0,Y 368.914,Z 152.532,A -85,B 0,C 180,E1 -12659.045,E2 -12659.045} C_VEL
LIN {X 0,Y 368.93,Z 152.61,A -85,B 0,C 180,E1 -12660.114,E2 -12660.114} C_VEL
LIN {X 0,Y 371.4,Z 164.031,A -85,B 0,C 180,E1 -12662.989,E2 -12662.989} C_VEL
LIN {X 0,Y 372.741,Z 171.639,A -85,B 0,C 180,E1 -12664.829,E2 -12664.829} C_VEL
LIN {X 0,Y 371.85,Z 182.361,A -85,B 0,C 180,E1 -12667.204,E2 -12667.204} C_VEL
LIN {X 0,Y 371.405,Z 187.463,A -85,B 0,C 180,E1 -12668.325,E2 -12668.325} C_VEL
LIN {X 0,Y 376.556,Z 219.295,A -85,B 0,C 180,E1 -12669.276,E2 -12669.276} C_VEL
LIN {X 0,Y 376.799,Z 225.06,A -85,B 0,C 180,E1 -12669.404,E2 -12669.404} C_VEL
LIN {X 0,Y 375.628,Z 296.162,A -85,B 0,C 180,E1 -12670.781,E2 -12670.781} C_VEL
LIN {X 0,Y 375.004,Z 309.377,A -85,B 0,C 180,E1 -12671.244,E2 -12671.244} C_VEL
LIN {X 0,Y 374.134,Z 321.511,A -85,B 0,C 180,E1 -12671.873,E2 -12671.873} C_VEL
LIN {X 0,Y 373.127,Z 333.762,A -85,B 0,C 180,E1 -12672.743,E2 -12672.743} C_VEL
LIN {X 0,Y 372,Z 345.355,A -85,B 0,C 180,E1 -12673.819,E2 -12673.819} C_VEL
LIN {X 0,Y 371.028,Z 355.671,A -85,B 0,C 180,E1 -12675.026,E2 -12675.026} C_VEL
LIN {X 0,Y 370.133,Z 364.343,A -85,B 0,C 180,E1 -12676.27,E2 -12676.27} C_VEL
LIN {X 0,Y 369.333,Z 372.229,A -85,B 0,C 180,E1 -12677.638,E2 -12677.638} C_VEL
LIN {X 0,Y 368.498,Z 379.93,A -85,B 0,C 180,E1 -12679.283,E2 -12679.283} C_VEL
LIN {X 0,Y 367.927,Z 387.041,A -85,B 0,C 180,E1 -12681.21,E2 -12681.21} C_VEL
LIN {X 0,Y 367.598,Z 391.772,A -85,B 0,C 180,E1 -12682.861,E2 -12682.861} C_VEL
LIN {X 0,Y 367.445,Z 395.391,A -85,B 0,C 180,E1 -12684.512,E2 -12684.512} C_VEL
LIN {X 0,Y 367.451,Z 397.26,A -85,B 0,C 180,E1 -12685.612,E2 -12685.612} C_VEL
LIN {X 0,Y 367.398,Z 399.658,A -85,B 0,C 180,E1 -12687.807,E2 -12687.807} C_VEL
LIN {X 0,Y 367.469,Z 400.271,A -85,B 0,C 180,E1 -12688.904,E2 -12688.904} C_VEL
LIN {X 0,Y 367.508,Z 400.487,A -85,B 0,C 180,E1 -12689.999,E2 -12689.999} C_VEL
LIN {X 0,Y 367.469,Z 400.267,A -85,B 0,C 180,E1 -12691.095,E2 -12691.095} C_VEL
LIN {X 0,Y 367.383,Z 398.65,A -85,B 0,C 180,E1 -12693.289,E2 -12693.289} C_VEL
LIN {X 0,Y 367.454,Z 397.248,A -85,B 0,C 180,E1 -12694.387,E2 -12694.387} C_VEL
LIN {X 0,Y 367.477,Z 394.351,A -85,B 0,C 180,E1 -12696.009,E2 -12696.009} C_VEL
LIN {X 0,Y 367.699,Z 390.307,A -85,B 0,C 180,E1 -12697.688,E2 -12697.688} C_VEL
LIN {X 0,Y 368.135,Z 384.175,A -85,B 0,C 180,E1 -12699.615,E2 -12699.615} C_VEL
LIN {X 0,Y 368.728,Z 377.48,A -85,B 0,C 180,E1 -12701.265,E2 -12701.265} C_VEL
LIN {X 0,Y 369.645,Z 369.183,A -85,B 0,C 180,E1 -12702.908,E2 -12702.908} C_VEL
LIN {X 0,Y 370.522,Z 360.677,A -85,B 0,C 180,E1 -12704.275,E2 -12704.275} C_VEL
LIN {X 0,Y 371.496,Z 350.167,A -85,B 0,C 180,E1 -12705.639,E2 -12705.639} C_VEL
LIN {X 0,Y 372.651,Z 338.346,A -85,B 0,C 180,E1 -12706.855,E2 -12706.855} C_VEL
LIN {X 0,Y 373.721,Z 326.455,A -85,B 0,C 180,E1 -12707.793,E2 -12707.793} C_VEL
LIN {X 0,Y 374.626,Z 314.082,A -85,B 0,C 180,E1 -12708.526,E2 -12708.526} C_VEL
LIN {X 0,Y 375.386,Z 301.37,A -85,B 0,C 180,E1 -12709.053,E2 -12709.053} C_VEL
LIN {X 0,Y 375.806,Z 288.008,A -85,B 0,C 180,E1 -12709.386,E2 -12709.386} C_VEL
LIN {X 0,Y 376.676,Z 220.43,A -85,B 0,C 180,E1 -12710.681,E2 -12710.681} C_VEL
LIN {X 0,Y 372.431,Z 193.471,A -85,B 0,C 180,E1 -12711.469,E2 -12711.469} C_VEL
LIN {X 0,Y 371.372,Z 187.494,A -85,B 0,C 180,E1 -12711.655,E2 -12711.655} C_VEL
LIN {X 0,Y 372.767,Z 172.294,A -85,B 0,C 180,E1 -12715.005,E2 -12715.005} C_VEL
LIN {X 0,Y 371.397,Z 163.963,A -85,B 0,C 180,E1 -12717.01,E2 -12717.01} C_VEL
LIN {X 0,Y 368.935,Z 152.532,A -85,B 0,C 180,E1 -12719.923,E2 -12719.923} C_VEL
LIN {X 0,Y 368.892,Z 152.537,A -85,B 0,C 180,E1 -12723.537,E2 -12723.537} C_VEL
LIN {X 0,Y 368.895,Z 152.531,A -85,B 0,C 180,E1 -12726.854,E2 -12726.854} C_VEL
LIN {X 0,Y 368.879,Z 152.532,A -85,B 0,C 180,E1 -12730.373,E2 -12730.373} C_VEL
LIN {X 0,Y 368.877,Z 152.535,A -85,B 0,C 180,E1 -12733.615,E2 -12733.615} C_VEL
LIN {X 0,Y 368.877,Z 152.534,A -85,B 0,C 180,E1 -12736.694,E2 -12736.694} C_VEL
LIN {X 0,Y 368.878,Z 152.534,A -85,B 0,C 180,E1 -12739.647,E2 -12739.647} C_VEL
LIN {X 0,Y 368.89,Z 152.536,A -85,B 0,C 180,E1 -12743.144,E2 -12743.144} C_VEL
LIN {X 0,Y 368.888,Z 152.533,A -85,B 0,C 180,E1 -12746.461,E2 -12746.461} C_VEL
LIN {X 0,Y 368.905,Z 152.533,A -85,B 0,C 180,E1 -12749.044,E2 -12749.044} C_VEL
LIN {X 0,Y 368.903,Z 152.53,A -85,B 0,C 180,E1 -12751.557,E2 -12751.557} C_VEL
LIN {X 0,Y 368.878,Z 152.534,A -85,B 0,C 180,E1 -12755.219,E2 -12755.219} C_VEL
LIN {X 0,Y 368.89,Z 152.531,A -85,B 0,C 180,E1 -12757.602,E2 -12757.602} C_VEL
LIN {X 0,Y 368.905,Z 152.53,A -85,B 0,C 180,E1 -12761.103,E2 -12761.103} C_VEL
LIN {X 0,Y 368.93,Z 152.531,A -85,B 0,C 180,E1 -12764.532,E2 -12764.532} C_VEL
LIN {X 0,Y 369.048,Z 152.513,A -85,B 0,C 180,E1 -12766.79,E2 -12766.79} C_VEL
LIN {X 0,Y 369.048,Z 152.517,A -85,B 0,C 180,E1 -12770.131,E2 -12770.131} C_VEL
LIN {X 0,Y 369.144,Z 152.5,A -85,B 0,C 180,E1 -12773.441,E2 -12773.441} C_VEL
LIN {X 0,Y 369.285,Z 152.486,A -85,B 0,C 180,E1 -12777.819,E2 -12777.819} C_VEL
LIN {X 0,Y 369.291,Z 152.484,A -85,B 0,C 180,E1 -12782.181,E2 -12782.181} C_VEL
LIN {X 0,Y 369.149,Z 152.499,A -85,B 0,C 180,E1 -12786.559,E2 -12786.559} C_VEL
LIN {X 0,Y 369.054,Z 152.515,A -85,B 0,C 180,E1 -12789.869,E2 -12789.869} C_VEL
LIN {X 0,Y 369.029,Z 152.518,A -85,B 0,C 180,E1 -12793.773,E2 -12793.773} C_VEL
LIN {X 0,Y 368.945,Z 152.528,A -85,B 0,C 180,E1 -12797.745,E2 -12797.745} C_VEL
LIN {X 0,Y 368.921,Z 152.532,A -85,B 0,C 180,E1 -12801.22,E2 -12801.22} C_VEL
LIN {X 0,Y 368.903,Z 152.531,A -85,B 0,C 180,E1 -12803.875,E2 -12803.875} C_VEL
LIN {X 0,Y 368.859,Z 152.541,A -85,B 0,C 180,E1 -12807.212,E2 -12807.212} C_VEL
LIN {X 0,Y 368.887,Z 152.533,A -85,B 0,C 180,E1 -12809.693,E2 -12809.693} C_VEL
LIN {X 0,Y 368.889,Z 152.538,A -85,B 0,C 180,E1 -12813.044,E2 -12813.044} C_VEL
LIN {X 0,Y 368.906,Z 152.529,A -85,B 0,C 180,E1 -12816.198,E2 -12816.198} C_VEL
LIN {X 0,Y 368.869,Z 152.539,A -85,B 0,C 180,E1 -12818.958,E2 -12818.958} C_VEL
LIN {X 0,Y 368.865,Z 152.534,A -85,B 0,C 180,E1 -12822.008,E2 -12822.008} C_VEL
LIN {X 0,Y 368.874,Z 152.535,A -85,B 0,C 180,E1 -12825.177,E2 -12825.177} C_VEL
LIN {X 0,Y 368.87,Z 152.535,A -85,B 0,C 180,E1 -12828.177,E2 -12828.177} C_VEL
LIN {X 0,Y 368.876,Z 152.533,A -85,B 0,C 180,E1 -12831.367,E2 -12831.367} C_VEL
LIN {X 0,Y 368.934,Z 152.526,A -85,B 0,C 180,E1 -12835.148,E2 -12835.148} C_VEL
LIN {X 0,Y 368.928,Z 152.527,A -85,B 0,C 180,E1 -12839.048,E2 -12839.048} C_VEL
LIN {X 0,Y 368.869,Z 152.535,A -85,B 0,C 180,E1 -12842.79,E2 -12842.79} C_VEL
LIN {X 0,Y 368.952,Z 152.652,A -85,B 0,C 180,E1 -12845.644,E2 -12845.644} C_VEL
LIN {X 0,Y 371.096,Z 162.923,A -85,B 0,C 180,E1 -12848.387,E2 -12848.387} C_VEL
LIN {X 0,Y 374.019,Z 171.419,A -85,B 0,C 180,E1 -12848.739,E2 -12848.739} C_VEL
LIN {X 0,Y 377.225,Z 187.351,A -85,B 0,C 180,E1 -12849.249,E2 -12849.249} C_VEL
LIN {X 0,Y 376.083,Z 265.031,A -85,B 0,C 180,E1 -12850.735,E2 -12850.735} C_VEL
LIN {X 0,Y 375.691,Z 277.935,A -85,B 0,C 180,E1 -12851.104,E2 -12851.104} C_VEL
LIN {X 0,Y 375.053,Z 291.177,A -85,B 0,C 180,E1 -12851.708,E2 -12851.708} C_VEL
LIN {X 0,Y 374.192,Z 303.562,A -85,B 0,C 180,E1 -12852.513,E2 -12852.513} C_VEL
LIN {X 0,Y 373.309,Z 314.654,A -85,B 0,C 180,E1 -12853.457,E2 -12853.457} C_VEL
LIN {X 0,Y 372.603,Z 324.311,A -85,B 0,C 180,E1 -12854.492,E2 -12854.492} C_VEL
LIN {X 0,Y 371.525,Z 334.109,A -85,B 0,C 180,E1 -12855.765,E2 -12855.765} C_VEL
LIN {X 0,Y 370.574,Z 342.596,A -85,B 0,C 180,E1 -12857.125,E2 -12857.125} C_VEL
LIN {X 0,Y 369.685,Z 350.838,A -85,B 0,C 180,E1 -12858.764,E2 -12858.764} C_VEL
LIN {X 0,Y 369.041,Z 356.477,A -85,B 0,C 180,E1 -12860.132,E2 -12860.132} C_VEL
LIN {X 0,Y 368.44,Z 361.971,A -85,B 0,C 180,E1 -12861.776,E2 -12861.776} C_VEL
LIN {X 0,Y 368.095,Z 366.279,A -85,B 0,C 180,E1 -12863.423,E2 -12863.423} C_VEL
LIN {X 0,Y 367.912,Z 368.559,A -85,B 0,C 180,E1 -12864.52,E2 -12864.52} C_VEL
LIN {X 0,Y 367.69,Z 370.417,A -85,B 0,C 180,E1 -12865.616,E2 -12865.616} C_VEL
LIN {X 0,Y 367.603,Z 371.812,A -85,B 0,C 180,E1 -12866.713,E2 -12866.713} C_VEL
LIN {X 0,Y 367.519,Z 373.416,A -85,B 0,C 180,E1 -12868.905,E2 -12868.905} C_VEL
LIN {X 0,Y 367.51,Z 373.648,A -85,B 0,C 180,E1 -12870.001,E2 -12870.001} C_VEL
LIN {X 0,Y 367.519,Z 373.459,A -85,B 0,C 180,E1 -12871.096,E2 -12871.096} C_VEL
LIN {X 0,Y 367.598,Z 371.912,A -85,B 0,C 180,E1 -12873.289,E2 -12873.289} C_VEL
LIN {X 0,Y 367.682,Z 370.56,A -85,B 0,C 180,E1 -12874.385,E2 -12874.385} C_VEL
LIN {X 0,Y 367.99,Z 367.697,A -85,B 0,C 180,E1 -12876.03,E2 -12876.03} C_VEL
LIN {X 0,Y 368.258,Z 363.821,A -85,B 0,C 180,E1 -12877.678,E2 -12877.678} C_VEL
LIN {X 0,Y 368.786,Z 358.815,A -85,B 0,C 180,E1 -12879.323,E2 -12879.323} C_VEL
LIN {X 0,Y 369.508,Z 352.509,A -85,B 0,C 180,E1 -12880.965,E2 -12880.965} C_VEL
LIN {X 0,Y 370.366,Z 344.615,A -85,B 0,C 180,E1 -12882.605,E2 -12882.605} C_VEL
LIN {X 0,Y 371.316,Z 336.563,A -85,B 0,C 180,E1 -12883.965,E2 -12883.965} C_VEL
LIN {X 0,Y 372.355,Z 326.736,A -85,B 0,C 180,E1 -12885.322,E2 -12885.322} C_VEL
LIN {X 0,Y 373.15,Z 317.07,A -85,B 0,C 180,E1 -12886.411,E2 -12886.411} C_VEL
LIN {X 0,Y 374.041,Z 306.6,A -85,B 0,C 180,E1 -12887.355,E2 -12887.355} C_VEL
LIN {X 0,Y 374.368,Z 301.75,A -85,B 0,C 180,E1 -12887.724,E2 -12887.724} C_VEL
LIN {X 0,Y 374.126,Z 296.441,A -85,B 0,C 180,E1 -12888.121,E2 -12888.121} C_VEL
LIN {X 0,Y 371.991,Z 287.703,A -85,B 0,C 180,E1 -12888.764,E2 -12888.764} C_VEL
LIN {X 0,Y 369.724,Z 278.713,A -85,B 0,C 180,E1 -12889.302,E2 -12889.302} C_VEL
LIN {X 0,Y 369.266,Z 273.016,A -85,B 0,C 180,E1 -12889.53,E2 -12889.53} C_VEL
LIN {X 0,Y 369.698,Z 252.733,A -85,B 0,C 180,E1 -12889.974,E2 -12889.974} C_VEL
LIN {X 0,Y 370.637,Z 188.059,A -85,B 0,C 180,E1 -12891.234,E2 -12891.234} C_VEL
